KUKA KRL program: MyProgram_324().src

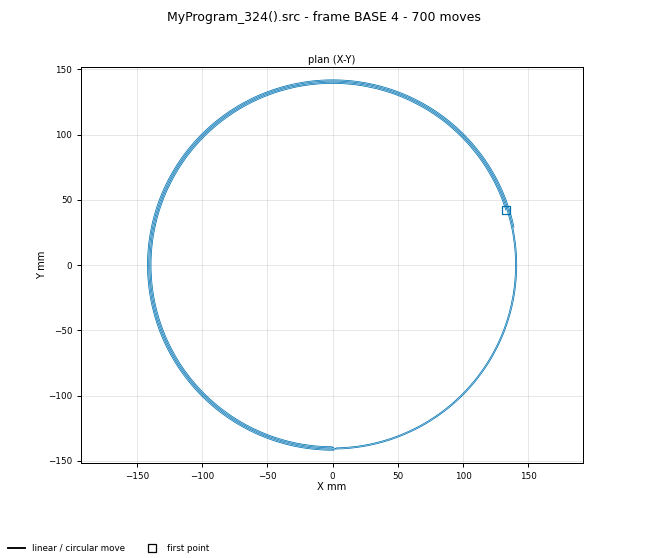
[picture p0: tool path of MyProgram_324().src in frame BASE 4, 700 of 700 moves have a stored position in this frame; points joined in program order, loops and branches not executed]
&ACCESS RVP
&REL 1
&PARAM TEMPLATE = C:\KRC\Roboter\Template\vorgabe
&PARAM EDITMASK = *
DEF MyProgram_324()
; ---- Setting reference (Base) ----
$BASE = BASE_DATA[4]

; --------------------------
; ---- Setting tool (TCP) ----
$TOOL = TOOL_DATA[3]
; --------------------------

$VEL.CP = VEL_APROX_PRINT
Startdeposition()
$VEL.CP = VEL_PRINT
LIN {X 132.7223,Y 42.0418,Z 186,A 20.4028,B 2.9301,C 0.1265,E1 3.0853,E2 432.9695} C_DIS
LIN {X 131.632,Y 45.3396,Z 186,A 21.7907,B 2.9303,C 0.1231,E1 3.0841,E2 431.5863} C_DIS
LIN {X 130.5462,Y 48.3787,Z 186,A 22.9188,B 2.9304,C 0.1215,E1 3.083,E2 430.4833} C_DIS
LIN {X 129.2167,Y 51.8236,Z 186,A 24.4942,B 2.9306,C 0.1169,E1 3.0814,E2 428.9} C_DIS
LIN {X 127.8365,Y 55.14,Z 186,A 25.9088,B 2.9307,C 0.1137,E1 3.0799,E2 427.493} C_DIS
LIN {X 126.4976,Y 58.1464,Z 186,A 27.093,B 2.9307,C 0.1118,E1 3.0786,E2 426.3301} C_DIS
LIN {X 124.9581,Y 61.3847,Z 186,A 28.6212,B 2.9309,C 0.1075,E1 3.0767,E2 424.7946} C_DIS
LIN {X 123.3471,Y 64.5607,Z 186,A 30.0105,B 2.9311,C 0.1045,E1 3.0749,E2 423.4145} C_DIS
LIN {X 121.2394,Y 68.4412,Z 186,A 31.8526,B 2.9312,C 0.0998,E1 3.0724,E2 421.5688} C_DIS
LIN {X 118.9409,Y 72.3624,Z 186,A 33.6675,B 2.9314,C 0.0957,E1 3.0698,E2 419.7604} C_DIS
LIN {X 116.4929,Y 76.2409,Z 186,A 35.4947,B 2.9314,C 0.0917,E1 3.0671,E2 417.9403} C_DIS
LIN {X 114.0875,Y 79.7952,Z 186,A 37.1739,B 2.9316,C 0.0884,E1 3.0644,E2 416.2718} C_DIS
LIN {X 111.3825,Y 83.5299,Z 186,A 38.922,B 2.9316,C 0.0853,E1 3.0616,E2 414.5422} C_DIS
LIN {X 105.7703,Y 90.5313,Z 186,A 42.3743,B 2.9318,C 0.0793,E1 3.0556,E2 411.1198} C_DIS
LIN {X 103.2392,Y 93.4068,Z 186,A 44.0814,B 2.932,C 0.0747,E1 3.0523,E2 409.3959} C_DIS
LIN {X 100.0339,Y 96.8315,Z 186,A 45.9143,B 2.932,C 0.0715,E1 3.0488,E2 407.575} C_DIS
LIN {X 96.6176,Y 100.241,Z 186,A 48.5902,B 2.9323,C 0.0615,E1 3.0433,E2 404.8112} C_DIS
LIN {X 91.8382,Y 104.6376,Z 186,A 50.3739,B 2.9323,C 0.064,E1 3.0398,E2 403.1402} C_DIS
LIN {X 88.2628,Y 107.67,Z 186,A 52.3174,B 2.9323,C 0.0602,E1 3.0356,E2 401.1947} C_DIS
LIN {X 84.6173,Y 110.5578,Z 186,A 54.1516,B 2.9323,C 0.0575,E1 3.0316,E2 399.3704} C_DIS
LIN {X 81.0366,Y 113.2086,Z 186,A 56.3803,B 2.9325,C 0.051,E1 3.0264,E2 397.0919} C_DIS
LIN {X 77.1098,Y 115.9192,Z 186,A 57.8819,B 2.9325,C 0.0516,E1 3.0231,E2 395.6486} C_DIS
LIN {X 73.3546,Y 118.3312,Z 186,A 59.6397,B 2.9325,C 0.0493,E1 3.019,E2 393.9008} C_DIS
LIN {X 69.3745,Y 120.7083,Z 186,A 61.5113,B 2.9325,C 0.0467,E1 3.0144,E2 392.0338} C_DIS
LIN {X 65.4235,Y 122.894,Z 186,A 63.1963,B 2.9325,C 0.0454,E1 3.0104,E2 390.3705} C_DIS
LIN {X 58.7576,Y 126.215,Z 186,A 66.3079,B 2.9326,C 0.0409,E1 3.0025,E2 387.2535} C_DIS
LIN {X 55.1898,Y 127.8149,Z 186,A 67.7185,B 2.9326,C 0.0405,E1 2.999,E2 385.8679} C_DIS
LIN {X 52.6155,Y 128.8975,Z 186,A 68.9895,B 2.9326,C 0.0382,E1 2.9957,E2 384.582} C_DIS
LIN {X 48.7864,Y 130.3935,Z 186,A 70.5342,B 2.9326,C 0.0374,E1 2.9917,E2 383.0558} C_DIS
LIN {X 45.2277,Y 131.6708,Z 186,A 72.3436,B 2.9327,C 0.0339,E1 2.9868,E2 381.2153} C_DIS
LIN {X 39.9443,Y 133.3707,Z 186,A 74.4722,B 2.9327,C 0.0329,E1 2.9812,E2 379.1066} C_DIS
LIN {X 36.2167,Y 134.4288,Z 186,A 75.8987,B 2.9327,C 0.0327,E1 2.9774,E2 377.7013} C_DIS
LIN {X 33.5088,Y 135.1309,Z 186,A 77.1314,B 2.9327,C 0.0312,E1 2.974,E2 376.4588} C_DIS
LIN {X 23.6749,Y 137.196,Z 186,A 81.8683,B 2.9328,C 0.0242,E1 2.9608,E2 371.6483} C_DIS
LIN {X 18.0755,Y 138.0433,Z 186,A 83.4414,B 2.9328,C 0.0283,E1 2.9567,E2 370.1703} C_DIS
LIN {X 14.3588,Y 138.4803,Z 186,A 85.0688,B 2.9328,C 0.027,E1 2.9522,E2 368.5327} C_DIS
LIN {X 10.3002,Y 138.8403,Z 186,A 86.6393,B 2.9328,C 0.027,E1 2.9478,E2 366.9759} C_DIS
LIN {X 7.1409,Y 139.0386,Z 186,A 87.9885,B 2.9328,C 0.0264,E1 2.9441,E2 365.6215} C_DIS
LIN {X 2.8453,Y 139.1938,Z 186,A 89.7701,B 2.9328,C 0.026,E1 2.9391,E2 363.8391} C_DIS
LIN {X -1.0873,Y 139.218,Z 186,A 91.4391,B 2.9328,C 0.0254,E1 2.9344,E2 362.1645} C_DIS
LIN {X -5.319,Y 139.1202,Z 186,A 92.8511,B 2.9328,C 0.0275,E1 2.9306,E2 360.794} C_DIS
LIN {X -10.208,Y 138.847,Z 186,A 95.1484,B 2.9328,C 0.0258,E1 2.9241,E2 358.4628} C_DIS
LIN {X -15.2684,Y 138.3824,Z 186,A 97.3365,B 2.9328,C 0.0255,E1 2.9179,E2 356.2638} C_DIS
LIN {X -18.8919,Y 137.9362,Z 186,A 98.9242,B 2.9328,C 0.0254,E1 2.9135,E2 354.6665} C_DIS
LIN {X -23.5933,Y 137.2096,Z 186,A 100.7482,B 2.9328,C 0.0268,E1 2.9085,E2 352.86} C_DIS
LIN {X -27.474,Y 136.4841,Z 186,A 102.3067,B 2.9328,C 0.0278,E1 2.9043,E2 351.3105} C_DIS
LIN {X -31.0328,Y 135.7188,Z 186,A 103.8636,B 2.9328,C 0.0282,E1 2.9,E2 349.7472} C_DIS
LIN {X -35.4652,Y 134.6291,Z 186,A 105.5281,B 2.9328,C 0.0305,E1 2.8956,E2 348.1102} C_DIS
LIN {X -38.2725,Y 133.8599,Z 186,A 107.0377,B 2.9328,C 0.0295,E1 2.8914,E2 346.5628} C_DIS
LIN {X -41.9969,Y 132.7366,Z 186,A 108.5373,B 2.9328,C 0.0312,E1 2.8874,E2 345.0766} C_DIS
LIN {X -45.3213,Y 131.6383,Z 186,A 110.2186,B 2.9328,C 0.0311,E1 2.8829,E2 343.3664} C_DIS
LIN {X -51.3729,Y 129.3983,Z 186,A 112.6899,B 2.9328,C 0.0344,E1 2.8765,E2 340.9196} C_DIS
LIN {X -54.8048,Y 127.9814,Z 186,A 114.2297,B 2.9327,C 0.0358,E1 2.8725,E2 339.3793} C_DIS
LIN {X -58.1767,Y 126.4836,Z 186,A 115.5667,B 2.9327,C 0.0384,E1 2.8692,E2 338.0656} C_DIS
LIN {X -60.9945,Y 125.1506,Z 186,A 117.3152,B 2.9327,C 0.0374,E1 2.8646,E2 336.2605} C_DIS
LIN {X -65.6557,Y 122.7702,Z 186,A 119.4155,B 2.9327,C 0.0403,E1 2.8595,E2 334.1683} C_DIS
LIN {X -69.1522,Y 120.8351,Z 186,A 121.2235,B 2.9327,C 0.0416,E1 2.855,E2 332.341} C_DIS
LIN {X -73.677,Y 118.1306,Z 186,A 123.2288,B 2.9326,C 0.0454,E1 2.8503,E2 330.3576} C_DIS
LIN {X -76.4881,Y 116.3301,Z 186,A 124.7057,B 2.9326,C 0.0469,E1 2.8468,E2 328.8689} C_DIS
LIN {X -80.3812,Y 113.675,Z 186,A 126.4295,B 2.9325,C 0.0508,E1 2.8429,E2 327.1733} C_DIS
LIN {X -85.7887,Y 109.6517,Z 186,A 129.4126,B 2.9325,C 0.0543,E1 2.8362,E2 324.1664} C_DIS
LIN {X -88.8265,Y 107.2052,Z 186,A 131.1719,B 2.9324,C 0.0564,E1 2.8323,E2 322.389} C_DIS
LIN {X -92.1361,Y 104.3746,Z 186,A 133.5756,B 2.9324,C 0.0569,E1 2.8271,E2 319.91} C_DIS
LIN {X -95.8456,Y 100.9798,Z 186,A 135.2159,B 2.9322,C 0.0626,E1 2.8239,E2 318.3252} C_DIS
LIN {X -98.943,Y 97.9462,Z 186,A 137.0176,B 2.9322,C 0.0659,E1 2.8203,E2 316.5226} C_DIS
LIN {X -102.1078,Y 94.6425,Z 186,A 138.7144,B 2.9321,C 0.0705,E1 2.8171,E2 314.8504} C_DIS
LIN {X -104.981,Y 91.4446,Z 186,A 140.7887,B 2.9321,C 0.0728,E1 2.8132,E2 312.7394} C_DIS
LIN {X -107.7815,Y 88.1264,Z 186,A 142.7152,B 2.9319,C 0.0761,E1 2.8097,E2 310.7967} C_DIS
LIN {X -110.7711,Y 84.3385,Z 186,A 144.7394,B 2.9319,C 0.0802,E1 2.8063,E2 308.7692} C_DIS
LIN {X -113.28,Y 80.9368,Z 186,A 146.8573,B 2.9318,C 0.0826,E1 2.8027,E2 306.6049} C_DIS
LIN {X -115.4664,Y 77.7861,Z 186,A 148.7724,B 2.9317,C 0.0849,E1 2.7997,E2 304.6482} C_DIS
LIN {X -118.3138,Y 73.3827,Z 186,A 150.3494,B 2.9315,C 0.0923,E1 2.7975,E2 303.1466} C_DIS
LIN {X -121.2066,Y 68.4995,Z 186,A 152.8996,B 2.9313,C 0.0971,E1 2.7938,E2 300.5712} C_DIS
LIN {X -123.0824,Y 65.0647,Z 186,A 154.5114,B 2.9312,C 0.101,E1 2.7917,E2 298.9603} C_DIS
LIN {X -124.7194,Y 61.8686,Z 186,A 156.0226,B 2.9311,C 0.1046,E1 2.7898,E2 297.4461} C_DIS
LIN {X -126.1022,Y 59.0017,Z 186,A 157.4751,B 2.931,C 0.1074,E1 2.7881,E2 295.9765} C_DIS
LIN {X -127.5991,Y 55.689,Z 186,A 158.8055,B 2.9308,C 0.1118,E1 2.7866,E2 294.6682} C_DIS
LIN {X -128.9832,Y 52.4027,Z 186,A 160.4995,B 2.9307,C 0.1148,E1 2.7847,E2 292.9466} C_DIS
LIN {X -130.2457,Y 49.1811,Z 186,A 162.0157,B 2.9305,C 0.1182,E1 2.7832,E2 291.4197} C_DIS
LIN {X -131.4915,Y 45.7449,Z 186,A 163.5273,B 2.9304,C 0.1221,E1 2.7818,E2 289.9083} C_DIS
LIN {X -132.4989,Y 42.741,Z 186,A 164.9566,B 2.9302,C 0.1252,E1 2.7805,E2 288.464} C_DIS
LIN {X -133.544,Y 39.3531,Z 186,A 166.487,B 2.9301,C 0.1288,E1 2.7793,E2 286.9256} C_DIS
LIN {X -134.4876,Y 35.9962,Z 186,A 167.975,B 2.9299,C 0.1325,E1 2.7782,E2 285.4318} C_DIS
LIN {X -135.4954,Y 32.0004,Z 186,A 169.8584,B 2.9297,C 0.1365,E1 2.7769,E2 283.5256} C_DIS
LIN {X -136.2453,Y 28.643,Z 186,A 171.4142,B 2.9296,C 0.1399,E1 2.776,E2 281.953} C_DIS
LIN {X -137.073,Y 24.3655,Z 186,A 173.1645,B 2.9293,C 0.145,E1 2.7751,E2 280.2093} C_DIS
LIN {X -137.8774,Y 19.304,Z 186,A 175.9731,B 2.9292,C 0.1485,E1 2.774,E2 277.3117} C_DIS
LIN {X -138.4947,Y 14.2251,Z 186,A 177.6797,B 2.9288,C 0.1558,E1 2.7735,E2 275.6584} C_DIS
LIN {X -138.8515,Y 10.1468,Z 186,A 179.1361,B 2.9285,C 0.1613,E1 2.7731,E2 274.2326} C_DIS
LIN {X -139.1571,Y 4.2614,Z 186,A -178.1292,B 2.9282,C 0.1671,E1 2.7728,E2 271.4597} C_DIS
LIN {X -139.1979,Y -2.5987,Z 186,A -175.1607,B 2.9277,C 0.1745,E1 2.7728,E2 268.4743} C_DIS
LIN {X -138.9299,Y -9.0223,Z 186,A -172.252,B 2.9273,C 0.181,E1 2.7732,E2 265.5331} C_DIS
LIN {X -138.4477,Y -14.6613,Z 186,A -169.9308,B 2.9269,C 0.1876,E1 2.7738,E2 263.2143} C_DIS
LIN {X -138.0238,Y -18.2243,Z 186,A -168.3737,B 2.9267,C 0.1914,E1 2.7743,E2 261.6475} C_DIS
LIN {X -137.1804,Y -23.7653,Z 186,A -165.8389,B 2.9263,C 0.197,E1 2.7755,E2 259.0843} C_DIS
LIN {X -136.3999,Y -27.8879,Z 186,A -164.1464,B 2.926,C 0.2018,E1 2.7764,E2 257.3971} C_DIS
LIN {X -135.6392,Y -31.3814,Z 186,A -162.4754,B 2.9257,C 0.2051,E1 2.7774,E2 255.7008} C_DIS
LIN {X -134.6193,Y -35.5023,Z 186,A -160.7508,B 2.9254,C 0.21,E1 2.7786,E2 253.98} C_DIS
LIN {X -133.6857,Y -38.8692,Z 186,A -159.2487,B 2.9251,C 0.2136,E1 2.7798,E2 252.4702} C_DIS
LIN {X -132.7391,Y -41.989,Z 186,A -157.9755,B 2.9249,C 0.2174,E1 2.7808,E2 251.2067} C_DIS
LIN {X -131.652,Y -45.2818,Z 186,A -156.5515,B 2.9246,C 0.2212,E1 2.7821,E2 249.7838} C_DIS
LIN {X -129.709,Y -50.5783,Z 186,A -153.8693,B 2.9242,C 0.2259,E1 2.7847,E2 247.0551} C_DIS
LIN {X -128.6254,Y -53.2752,Z 186,A -152.4667,B 2.924,C 0.2282,E1 2.7863,E2 245.6256} C_DIS
LIN {X -126.553,Y -58.0266,Z 186,A -150.3996,B 2.9236,C 0.2338,E1 2.7886,E2 243.5682} C_DIS
LIN {X -125.0099,Y -61.2796,Z 186,A -148.8804,B 2.9233,C 0.2374,E1 2.7904,E2 242.0446} C_DIS
LIN {X -123.6519,Y -63.9802,Z 186,A -147.5183,B 2.9231,C 0.24,E1 2.7922,E2 240.6673} C_DIS
LIN {X -119.8995,Y -70.7624,Z 186,A -144.2009,B 2.9225,C 0.2471,E1 2.7968,E2 237.3341} C_DIS
LIN {X -117.3139,Y -74.9705,Z 186,A -142.0411,B 2.9221,C 0.2513,E1 2.8,E2 235.158} C_DIS
LIN {X -114.7566,Y -78.8292,Z 186,A -140.0835,B 2.9218,C 0.2554,E1 2.8031,E2 233.1939} C_DIS
LIN {X -112.8116,Y -81.5885,Z 186,A -138.2374,B 2.9217,C 0.2565,E1 2.8062,E2 231.2867} C_DIS
LIN {X -110.2703,Y -84.9925,Z 186,A -136.7891,B 2.9212,C 0.2616,E1 2.8086,E2 229.8793} C_DIS
LIN {X -107.4976,Y -88.4735,Z 186,A -134.8803,B 2.9209,C 0.2651,E1 2.8119,E2 227.9605} C_DIS
LIN {X -104.5729,Y -91.9119,Z 186,A -133.2398,B 2.9205,C 0.2699,E1 2.8149,E2 226.3495} C_DIS
LIN {X -102.4762,Y -94.243,Z 186,A -131.6371,B 2.9204,C 0.271,E1 2.818,E2 224.705} C_DIS
LIN {X -99.0053,Y -97.8835,Z 186,A -129.2575,B 2.9201,C 0.2735,E1 2.8227,E2 222.284} C_DIS
LIN {X -96.5135,Y -100.3416,Z 186,A -127.9872,B 2.9198,C 0.277,E1 2.8252,E2 221.0369} C_DIS
LIN {X -93.1987,Y -103.4277,Z 186,A -126.0443,B 2.9195,C 0.28,E1 2.8292,E2 219.0834} C_DIS
LIN {X -89.6587,Y -106.5105,Z 186,A -124.0623,B 2.9192,C 0.283,E1 2.8335,E2 217.0948} C_DIS
LIN {X -86,Y -109.4857,Z 186,A -122.1302,B 2.9189,C 0.2863,E1 2.8377,E2 215.164} C_DIS
LIN {X -77.5113,Y -115.6511,Z 186,A -117.9132,B 2.9182,C 0.2934,E1 2.8472,E2 210.961} C_DIS
LIN {X -74.5846,Y -117.5601,Z 186,A -116.1603,B 2.9182,C 0.2937,E1 2.8514,E2 209.1654} C_DIS
LIN {X -70.7202,Y -119.9243,Z 186,A -114.2581,B 2.918,C 0.2959,E1 2.856,E2 207.2579} C_DIS
LIN {X -66.4872,Y -122.3218,Z 186,A -111.2975,B 2.9183,C 0.2929,E1 2.8636,E2 204.1656} C_DIS
LIN {X -60.0963,Y -125.5826,Z 186,A -109.3331,B 2.9174,C 0.3018,E1 2.8682,E2 202.3365} C_DIS
LIN {X -56.0089,Y -127.4608,Z 186,A -107.4407,B 2.9172,C 0.3034,E1 2.873,E2 200.4383} C_DIS
LIN {X -52.4435,Y -128.9668,Z 186,A -105.8095,B 2.9171,C 0.3047,E1 2.8773,E2 198.8016} C_DIS
LIN {X -48.4538,Y -130.5181,Z 186,A -103.8163,B 2.9171,C 0.3047,E1 2.8826,E2 196.7763} C_DIS
LIN {X -44.2579,Y -131.9997,Z 186,A -102.3244,B 2.9167,C 0.3082,E1 2.8864,E2 195.3304} C_DIS
LIN {X -41.04,Y -133.0354,Z 186,A -100.7788,B 2.9167,C 0.3082,E1 2.8906,E2 193.7634} C_DIS
LIN {X -37.7743,Y -133.9992,Z 186,A -99.5511,B 2.9165,C 0.3102,E1 2.8938,E2 192.559} C_DIS
LIN {X -34.537,Y -134.8699,Z 186,A -97.2089,B 2.917,C 0.3048,E1 2.9005,E2 190.0842} C_DIS
LIN {X -28.8904,Y -136.1919,Z 186,A -95.4264,B 2.9165,C 0.3097,E1 2.9051,E2 188.3843} C_DIS
LIN {X -23.7358,Y -137.1857,Z 186,A -93.3501,B 2.9164,C 0.311,E1 2.9108,E2 186.3188} C_DIS
LIN {X -19.9134,Y -137.7903,Z 186,A -91.8953,B 2.9163,C 0.3123,E1 2.9148,E2 184.8822} C_DIS
LIN {X -16.6105,Y -138.2273,Z 186,A -90.3853,B 2.9163,C 0.3116,E1 2.919,E2 183.3527} C_DIS
LIN {X -13.0475,Y -138.6092,Z 186,A -88.8614,B 2.9163,C 0.3115,E1 2.9233,E2 181.8214} C_DIS
LIN {X -8.7396,Y -138.9473,Z 186,A -87.083,B 2.9163,C 0.3115,E1 2.9283,E2 180.0424} C_DIS
LIN {X -4.337,Y -139.155,Z 186,A -85.2848,B 2.9163,C 0.3115,E1 2.9333,E2 178.2455} C_DIS
LIN {X -0.6821,Y -139.2202,Z 186,A -83.7898,B 2.9163,C 0.3113,E1 2.9375,E2 176.7511} C_DIS
LIN {X -0.6821,Y -139.2202,Z 186,A -83.7898,B 2.9163,C 0.3113,E1 2.9375,E2 176.7511} C_DIS
Enddeposition()
LIN {X 1.0073,Y -140.1176,Z 186,A -83.0914,B 2.892,C 0.3118,E1 2.9151,E2 176.0888} C_DIS
Startdeposition()
$VEL.CP = VEL_PRINT
LIN {X -2.8203,Y -140.0942,Z 186,A -85.3593,B 2.8914,C 0.317,E1 2.9085,E2 178.4541} C_DIS
LIN {X -7.0046,Y -139.9465,Z 186,A -86.9368,B 2.8915,C 0.3162,E1 2.9041,E2 180.014} C_DIS
LIN {X -10.1238,Y -139.7554,Z 186,A -88.277,B 2.8915,C 0.3166,E1 2.9004,E2 181.3632} C_DIS
LIN {X -14.2012,Y -139.4023,Z 186,A -90.0662,B 2.8915,C 0.3172,E1 2.8953,E2 183.169} C_DIS
LIN {X -18.1624,Y -138.9394,Z 186,A -91.5726,B 2.8915,C 0.3161,E1 2.8912,E2 184.659} C_DIS
LIN {X -21.6584,Y -138.4377,Z 186,A -93.0477,B 2.8915,C 0.316,E1 2.8871,E2 186.1389} C_DIS
LIN {X -26.4802,Y -137.5967,Z 186,A -95.0602,B 2.8916,C 0.3154,E1 2.8816,E2 188.1536} C_DIS
LIN {X -30.6439,Y -136.7307,Z 186,A -97.0086,B 2.8916,C 0.316,E1 2.8762,E2 190.1311} C_DIS
LIN {X -38.0299,Y -134.8621,Z 186,A -99.9566,B 2.8919,C 0.3133,E1 2.8683,E2 193.0572} C_DIS
LIN {X -42.2307,Y -133.6066,Z 186,A -101.7675,B 2.8919,C 0.3122,E1 2.8634,E2 194.8711} C_DIS
LIN {X -49.1907,Y -131.203,Z 186,A -104.7675,B 2.8922,C 0.3098,E1 2.8555,E2 197.8703} C_DIS
LIN {X -52.5755,Y -129.8838,Z 186,A -106.3058,B 2.8923,C 0.3088,E1 2.8515,E2 199.4161} C_DIS
LIN {X -55.9211,Y -128.4791,Z 186,A -107.8545,B 2.8924,C 0.3078,E1 2.8475,E2 200.9739} C_DIS
LIN {X -59.073,Y -127.0606,Z 186,A -109.2324,B 2.8926,C 0.3062,E1 2.844,E2 202.3472} C_DIS
LIN {X -61.9775,Y -125.6691,Z 186,A -110.9944,B 2.8926,C 0.3072,E1 2.8394,E2 204.1697} C_DIS
LIN {X -65.5403,Y -123.8491,Z 186,A -112.3239,B 2.8929,C 0.3036,E1 2.8362,E2 205.458} C_DIS
LIN {X -69.6738,Y -121.5736,Z 186,A -114.3235,B 2.8931,C 0.3016,E1 2.8313,E2 207.4673} C_DIS
LIN {X -73.6489,Y -119.2079,Z 186,A -116.2465,B 2.8933,C 0.2993,E1 2.8267,E2 209.3948} C_DIS
LIN {X -77.3828,Y -116.8184,Z 186,A -118.1408,B 2.8936,C 0.2972,E1 2.8222,E2 211.3001} C_DIS
LIN {X -82.8133,Y -113.0326,Z 186,A -121.0194,B 2.8939,C 0.294,E1 2.8156,E2 214.2019} C_DIS
LIN {X -86.9995,Y -109.8439,Z 186,A -123.1378,B 2.8942,C 0.2904,E1 2.811,E2 216.3157} C_DIS
LIN {X -90.5099,Y -106.9698,Z 186,A -125.2597,B 2.8944,C 0.2885,E1 2.8063,E2 218.4735} C_DIS
LIN {X -93.182,Y -104.6507,Z 186,A -126.5493,B 2.8948,C 0.2853,E1 2.8037,E2 219.7417} C_DIS
LIN {X -99.3475,Y -98.8158,Z 186,A -130.0753,B 2.8953,C 0.2791,E1 2.7966,E2 223.2747} C_DIS
LIN {X -102.3742,Y -95.6769,Z 186,A -131.9754,B 2.8956,C 0.2762,E1 2.7929,E2 225.1904} C_DIS
LIN {X -106.548,Y -91.0061,Z 186,A -134.4714,B 2.8961,C 0.2707,E1 2.7883,E2 227.6771} C_DIS
LIN {X -108.9363,Y -88.133,Z 186,A -137.1963,B 2.896,C 0.2727,E1 2.7833,E2 230.5608} C_DIS
LIN {X -113.5466,Y -82.1078,Z 186,A -139.3898,B 2.8969,C 0.262,E1 2.7798,E2 232.6331} C_DIS
LIN {X -116.1588,Y -78.3689,Z 186,A -141.3574,B 2.8973,C 0.2583,E1 2.7767,E2 234.6139} C_DIS
LIN {X -118.6593,Y -74.5284,Z 186,A -143.1364,B 2.8977,C 0.2536,E1 2.774,E2 236.3797} C_DIS
LIN {X -120.5144,Y -71.4903,Z 186,A -145.0644,B 2.8978,C 0.252,E1 2.7711,E2 238.3701} C_DIS
LIN {X -122.2481,Y -68.4828,Z 186,A -146.4171,B 2.8981,C 0.2484,E1 2.7693,E2 239.7134} C_DIS
LIN {X -124.3266,Y -64.6308,Z 186,A -148.2148,B 2.8985,C 0.244,E1 2.767,E2 241.5115} C_DIS
LIN {X -126.3123,Y -60.6565,Z 186,A -150.0063,B 2.8989,C 0.2394,E1 2.7647,E2 243.299} C_DIS
LIN {X -127.8057,Y -57.4429,Z 186,A -151.6407,B 2.8991,C 0.2365,E1 2.7628,E2 244.9572} C_DIS
LIN {X -129.3909,Y -53.7772,Z 186,A -153.1363,B 2.8995,C 0.2318,E1 2.7612,E2 246.4339} C_DIS
LIN {X -130.9844,Y -49.7724,Z 186,A -155.3764,B 2.8997,C 0.229,E1 2.7589,E2 248.7362} C_DIS
LIN {X -132.1779,Y -46.5121,Z 186,A -156.4594,B 2.9001,C 0.224,E1 2.7579,E2 249.7743} C_DIS
LIN {X -133.0781,Y -43.8676,Z 186,A -157.7354,B 2.9003,C 0.2215,E1 2.7568,E2 251.0675} C_DIS
LIN {X -134.2034,Y -40.2984,Z 186,A -159.4915,B 2.9006,C 0.2183,E1 2.7553,E2 252.8525} C_DIS
LIN {X -135.3756,Y -36.1585,Z 186,A -161.2152,B 2.9009,C 0.2134,E1 2.754,E2 254.5705} C_DIS
LIN {X -136.2522,Y -32.7009,Z 186,A -162.7135,B 2.9012,C 0.2096,E1 2.753,E2 256.0733} C_DIS
LIN {X -137.0113,Y -29.3591,Z 186,A -164.2143,B 2.9015,C 0.2061,E1 2.7521,E2 257.5864} C_DIS
LIN {X -137.8186,Y -25.307,Z 186,A -166.7114,B 2.9015,C 0.2043,E1 2.7508,E2 260.1875} C_DIS
LIN {X -138.7087,Y -19.8477,Z 186,A -168.0276,B 2.9022,C 0.1947,E1 2.7503,E2 261.3795} C_DIS
LIN {X -139.1085,Y -16.8203,Z 186,A -170.2463,B 2.9022,C 0.1946,E1 2.7495,E2 263.7236} C_DIS
LIN {X -139.6024,Y -12.0542,Z 186,A -171.4913,B 2.9028,C 0.1867,E1 2.7492,E2 264.8749} C_DIS
LIN {X -140.0378,Y -4.8813,Z 186,A -174.7473,B 2.9032,C 0.1795,E1 2.7487,E2 268.1706} C_DIS
LIN {X -140.114,Y -1.6302,Z 186,A -176.6869,B 2.9033,C 0.1778,E1 2.7486,E2 270.188} C_DIS
LIN {X -140.1002,Y 2.4604,Z 186,A -177.8971,B 2.9037,C 0.1716,E1 2.7486,E2 271.3376} C_DIS
LIN {X -139.7549,Y 10.1308,Z 186,A 178.8114,B 2.9042,C 0.1633,E1 2.7491,E2 274.6468} C_DIS
LIN {X -138.9275,Y 18.2534,Z 186,A 174.7575,B 2.9046,C 0.1563,E1 2.7504,E2 278.7901} C_DIS
LIN {X -138.3187,Y 22.4138,Z 186,A 173.4853,B 2.9049,C 0.15,E1 2.7509,E2 280.0041} C_DIS
LIN {X -137.5893,Y 26.5188,Z 186,A 171.6337,B 2.9051,C 0.1458,E1 2.7518,E2 281.8732} C_DIS
LIN {X -136.4611,Y 31.824,Z 186,A 169.3535,B 2.9054,C 0.1399,E1 2.7532,E2 284.1598} C_DIS
LIN {X -135.8128,Y 34.4801,Z 186,A 168.0816,B 2.9055,C 0.1374,E1 2.754,E2 285.4506} C_DIS
LIN {X -134.8776,Y 37.9746,Z 186,A 166.561,B 2.9057,C 0.1335,E1 2.7552,E2 286.9753} C_DIS
LIN {X -133.8797,Y 41.356,Z 186,A 165.0431,B 2.9059,C 0.1299,E1 2.7564,E2 288.5019} C_DIS
LIN {X -132.8695,Y 44.4938,Z 186,A 163.5863,B 2.906,C 0.1267,E1 2.7577,E2 289.9716} C_DIS
LIN {X -131.6328,Y 48.0318,Z 186,A 162.0329,B 2.9062,C 0.1227,E1 2.7591,E2 291.5265} C_DIS
LIN {X -130.5108,Y 50.9993,Z 186,A 160.6348,B 2.9062,C 0.1197,E1 2.7605,E2 292.9363} C_DIS
LIN {X -129.1805,Y 54.281,Z 186,A 159.1523,B 2.9064,C 0.1161,E1 2.7621,E2 294.4222} C_DIS
LIN {X -127.7897,Y 57.4787,Z 186,A 157.6404,B 2.9066,C 0.1127,E1 2.7638,E2 295.9439} C_DIS
LIN {X -126.244,Y 60.7995,Z 186,A 156.093,B 2.9067,C 0.1091,E1 2.7657,E2 297.4964} C_DIS
LIN {X -124.7604,Y 63.7873,Z 186,A 154.6494,B 2.9068,C 0.106,E1 2.7675,E2 298.949} C_DIS
LIN {X -123.0275,Y 67.0726,Z 186,A 152.9761,B 2.9069,C 0.1028,E1 2.7698,E2 300.6406} C_DIS
LIN {X -120.9497,Y 70.7512,Z 186,A 151.3206,B 2.9071,C 0.0984,E1 2.772,E2 302.2858} C_DIS
LIN {X -119.0618,Y 73.8837,Z 186,A 149.0959,B 2.9071,C 0.0976,E1 2.7755,E2 304.6004} C_DIS
LIN {X -116.3995,Y 78.0105,Z 186,A 147.5398,B 2.9073,C 0.0912,E1 2.7778,E2 306.0987} C_DIS
LIN {X -114.4773,Y 80.8049,Z 186,A 146.1663,B 2.9074,C 0.088,E1 2.7799,E2 307.4694} C_DIS
LIN {X -112.085,Y 84.0928,Z 186,A 144.4493,B 2.9075,C 0.0846,E1 2.7828,E2 309.1921} C_DIS
LIN {X -109.706,Y 87.1728,Z 186,A 142.4375,B 2.9075,C 0.0828,E1 2.7864,E2 311.2549} C_DIS
LIN {X -107.4678,Y 89.9177,Z 186,A 140.3627,B 2.9075,C 0.0822,E1 2.7903,E2 313.4059} C_DIS
LIN {X -103.1556,Y 94.8336,Z 186,A 138.8315,B 2.9079,C 0.0721,E1 2.7929,E2 314.7937} C_DIS
LIN {X -99.7013,Y 98.4597,Z 186,A 136.251,B 2.9079,C 0.0703,E1 2.798,E2 317.4391} C_DIS
LIN {X -96.4124,Y 101.6822,Z 186,A 134.12,B 2.9079,C 0.0678,E1 2.8023,E2 319.5994} C_DIS
LIN {X -93.9584,Y 103.9533,Z 186,A 133.0252,B 2.9081,C 0.0641,E1 2.8045,E2 320.6595} C_DIS
LIN {X -90.9705,Y 106.5783,Z 186,A 131.2328,B 2.9081,C 0.062,E1 2.8083,E2 322.4712} C_DIS
LIN {X -87.5,Y 109.4455,Z 186,A 129.3243,B 2.9081,C 0.0592,E1 2.8125,E2 324.3868} C_DIS
LIN {X -83.0265,Y 112.8765,Z 186,A 127.0447,B 2.9082,C 0.0553,E1 2.8176,E2 326.6615} C_DIS
LIN {X -80.4773,Y 114.7084,Z 186,A 125.6391,B 2.9082,C 0.0539,E1 2.8208,E2 328.0814} C_DIS
LIN {X -76.0708,Y 117.6767,Z 186,A 123.523,B 2.9083,C 0.0505,E1 2.8257,E2 330.189} C_DIS
LIN {X -69.6537,Y 121.585,Z 186,A 120.5702,B 2.9084,C 0.0457,E1 2.8327,E2 333.1251} C_DIS
LIN {X -66.865,Y 123.1407,Z 186,A 118.9491,B 2.9084,C 0.0457,E1 2.8368,E2 334.7842} C_DIS
LIN {X -63.6921,Y 124.8089,Z 186,A 116.8207,B 2.9084,C 0.0472,E1 2.8423,E2 336.9926} C_DIS
LIN {X -58.6521,Y 127.2552,Z 186,A 115.2003,B 2.9084,C 0.0413,E1 2.8462,E2 338.5297} C_DIS
LIN {X -55.5464,Y 128.6411,Z 186,A 113.3543,B 2.9084,C 0.0422,E1 2.8511,E2 340.4305} C_DIS
LIN {X -51.6471,Y 130.258,Z 186,A 112.0559,B 2.9085,C 0.0384,E1 2.8543,E2 341.6756} C_DIS
LIN {X -45.7089,Y 132.4564,Z 186,A 109.4422,B 2.9085,C 0.0363,E1 2.8612,E2 344.2907} C_DIS
LIN {X -42.6797,Y 133.4631,Z 186,A 108.0307,B 2.9085,C 0.0359,E1 2.8649,E2 345.7145} C_DIS
LIN {X -38.6935,Y 134.6748,Z 186,A 105.9805,B 2.9085,C 0.0367,E1 2.8706,E2 347.8062} C_DIS
LIN {X -35.0744,Y 135.6619,Z 186,A 104.8968,B 2.9085,C 0.0333,E1 2.8733,E2 348.8339} C_DIS
LIN {X -31.1063,Y 136.625,Z 186,A 103.121,B 2.9085,C 0.033,E1 2.8782,E2 350.6218} C_DIS
LIN {X -27.6399,Y 137.3686,Z 186,A 101.6275,B 2.9085,C 0.0326,E1 2.8823,E2 352.1198} C_DIS
LIN {X -19.4073,Y 138.7716,Z 186,A 98.2081,B 2.9085,C 0.0315,E1 2.8918,E2 355.5382} C_DIS
LIN {X -15.2807,Y 139.2861,Z 186,A 96.3935,B 2.9085,C 0.0319,E1 2.8968,E2 357.3659} C_DIS
LIN {X -9.1316,Y 139.8247,Z 186,A 94.0918,B 2.9086,C 0.0303,E1 2.9032,E2 359.6392} C_DIS
LIN {X -5.475,Y 140.0147,Z 186,A 92.504,B 2.9086,C 0.0308,E1 2.9076,E2 361.2375} C_DIS
LIN {X -1.7806,Y 140.1115,Z 186,A 90.8716,B 2.9086,C 0.0317,E1 2.9122,E2 362.8841} C_DIS
LIN {X 2.2977,Y 140.1029,Z 186,A 89.283,B 2.9086,C 0.0315,E1 2.9166,E2 364.4623} C_DIS
LIN {X 6.5026,Y 139.9717,Z 186,A 87.5403,B 2.9086,C 0.032,E1 2.9215,E2 366.2072} C_DIS
LIN {X 10.1851,Y 139.7509,Z 186,A 86.1055,B 2.9086,C 0.032,E1 2.9255,E2 367.6322} C_DIS
LIN {X 13.5142,Y 139.4684,Z 186,A 84.7785,B 2.9086,C 0.0323,E1 2.9292,E2 368.954} C_DIS
LIN {X 16.8125,Y 139.1094,Z 186,A 83.3856,B 2.9086,C 0.0331,E1 2.933,E2 370.3509} C_DIS
LIN {X 20.7808,Y 138.5735,Z 186,A 81.6286,B 2.9086,C 0.0348,E1 2.938,E2 372.122} C_DIS
LIN {X 24.9414,Y 137.8841,Z 186,A 80.0662,B 2.9086,C 0.0348,E1 2.9422,E2 373.6639} C_DIS
LIN {X 28.7642,Y 137.1389,Z 186,A 78.398,B 2.9086,C 0.0364,E1 2.9468,E2 375.341} C_DIS
LIN {X 34.8216,Y 135.7261,Z 186,A 76.0373,B 2.9086,C 0.037,E1 2.9532,E2 377.6786} C_DIS
LIN {X 37.7562,Y 134.9387,Z 186,A 74.7605,B 2.9086,C 0.0384,E1 2.9566,E2 378.9593} C_DIS
LIN {X 41.0365,Y 133.9775,Z 186,A 72.7793,B 2.9084,C 0.0439,E1 2.9621,E2 381.0117} C_DIS
LIN {X 45.9497,Y 132.3729,Z 186,A 71.3347,B 2.9084,C 0.0412,E1 2.9657,E2 382.3738} C_DIS
LIN {X 49.3723,Y 131.135,Z 186,A 69.8501,B 2.9084,C 0.0427,E1 2.9696,E2 383.8578} C_DIS
LIN {X 52.5122,Y 129.9093,Z 186,A 68.4786,B 2.9084,C 0.0443,E1 2.9732,E2 385.2282} C_DIS
LIN {X 55.9067,Y 128.4853,Z 186,A 67.0199,B 2.9084,C 0.0458,E1 2.9769,E2 386.6809} C_DIS
LIN {X 59.6622,Y 126.7873,Z 186,A 64.9469,B 2.9084,C 0.0509,E1 2.9823,E2 388.8016} C_DIS
LIN {X 63.296,Y 125.0105,Z 186,A 63.7666,B 2.9084,C 0.0495,E1 2.9851,E2 389.9232} C_DIS
LIN {X 66.2429,Y 123.4762,Z 186,A 62.3458,B 2.9083,C 0.0519,E1 2.9886,E2 391.3517} C_DIS
LIN {X 70.384,Y 121.1636,Z 186,A 60.4785,B 2.9083,C 0.0542,E1 2.9931,E2 393.2099} C_DIS
LIN {X 74.0809,Y 118.9391,Z 186,A 58.7482,B 2.9083,C 0.0567,E1 2.9972,E2 394.9359} C_DIS
LIN {X 77.9035,Y 116.4713,Z 186,A 56.7162,B 2.9081,C 0.0612,E1 3.002,E2 396.9892} C_DIS
LIN {X 80.7684,Y 114.5031,Z 186,A 55.59,B 2.9081,C 0.0612,E1 3.0045,E2 398.0788} C_DIS
LIN {X 84.2612,Y 111.9579,Z 186,A 53.8305,B 2.9081,C 0.0642,E1 3.0085,E2 399.8374} C_DIS
LIN {X 87.7944,Y 109.2093,Z 186,A 52.0517,B 2.908,C 0.0671,E1 3.0124,E2 401.6098} C_DIS
LIN {X 90.5408,Y 106.9436,Z 186,A 50.6985,B 2.908,C 0.069,E1 3.0152,E2 402.9503} C_DIS
LIN {X 94.7809,Y 103.204,Z 186,A 48.2327,B 2.9078,C 0.0748,E1 3.0204,E2 405.4356} C_DIS
LIN {X 97.2214,Y 100.9089,Z 186,A 47.0627,B 2.9078,C 0.0758,E1 3.0227,E2 406.5808} C_DIS
LIN {X 100.4442,Y 97.7014,Z 186,A 45.2766,B 2.9077,C 0.079,E1 3.0262,E2 408.358} C_DIS
LIN {X 103.505,Y 94.4529,Z 186,A 43.4994,B 2.9076,C 0.0825,E1 3.0296,E2 410.1295} C_DIS
LIN {X 105.9389,Y 91.7146,Z 186,A 42.0828,B 2.9076,C 0.085,E1 3.0321,E2 411.5362} C_DIS
LIN {X 109.786,Y 87.0711,Z 186,A 39.7594,B 2.9074,C 0.0893,E1 3.0362,E2 413.8421} C_DIS
LIN {X 112.085,Y 84.0928,Z 186,A 38.2173,B 2.9073,C 0.0928,E1 3.0388,E2 415.3851} C_DIS
LIN {X 114.795,Y 80.3539,Z 186,A 36.3996,B 2.9072,C 0.0966,E1 3.0418,E2 417.1945} C_DIS
LIN {X 117.3488,Y 76.5759,Z 186,A 34.6076,B 2.907,C 0.1004,E1 3.0445,E2 418.9778} C_DIS
LIN {X 119.8062,Y 72.6706,Z 186,A 32.8142,B 2.9069,C 0.1041,E1 3.0471,E2 420.76} C_DIS
LIN {X 122.1328,Y 68.6883,Z 186,A 31.0315,B 2.9068,C 0.1078,E1 3.0496,E2 422.5301} C_DIS
LIN {X 124.2212,Y 64.8315,Z 186,A 29.4036,B 2.9067,C 0.1108,E1 3.0517,E2 424.1375} C_DIS
LIN {X 125.8531,Y 61.6045,Z 186,A 27.9865,B 2.9065,C 0.1139,E1 3.0535,E2 425.5473} C_DIS
LIN {X 127.2965,Y 58.5628,Z 186,A 26.646,B 2.9065,C 0.1171,E1 3.055,E2 426.8837} C_DIS
LIN {X 128.7275,Y 55.3466,Z 186,A 25.2431,B 2.9063,C 0.1205,E1 3.0566,E2 428.2826} C_DIS
LIN {X 130.4291,Y 51.2095,Z 186,A 23.4905,B 2.9061,C 0.1246,E1 3.0584,E2 430.0262} C_DIS
LIN {X 131.7711,Y 47.6481,Z 186,A 22.0604,B 2.906,C 0.1276,E1 3.0598,E2 431.4407} C_DIS
LIN {X 132.8864,Y 44.4432,Z 186,A 20.6842,B 2.9058,C 0.1312,E1 3.061,E2 432.8162} C_DIS
LIN {X 134.0315,Y 40.86,Z 186,A 19.2077,B 2.9056,C 0.1347,E1 3.0623,E2 434.2855} C_DIS
LIN {X 135.6796,Y 35.0046,Z 186,A 16.9816,B 2.9054,C 0.139,E1 3.0639,E2 436.4792} C_DIS
LIN {X 136.5324,Y 31.512,Z 186,A 15.1481,B 2.9051,C 0.1465,E1 3.0651,E2 438.3603} C_DIS
LIN {X 137.2928,Y 28.0124,Z 186,A 13.7177,B 2.9049,C 0.1502,E1 3.0659,E2 439.7871} C_DIS
LIN {X 138.0122,Y 24.2255,Z 186,A 12.4853,B 2.9049,C 0.1513,E1 3.0665,E2 440.976} C_DIS
LIN {X 138.7697,Y 19.4206,Z 186,A 10.558,B 2.9046,C 0.1563,E1 3.0673,E2 442.8965} C_DIS
LIN {X 139.3092,Y 15.0667,Z 186,A 8.9556,B 2.9044,C 0.1594,E1 3.0678,E2 444.4751} C_DIS
LIN {X 139.675,Y 11.1945,Z 186,A 7.326,B 2.9041,C 0.1643,E1 3.0682,E2 446.1108} C_DIS
LIN {X 139.943,Y 7.0726,Z 186,A 5.816,B 2.9039,C 0.1673,E1 3.0684,E2 447.5985} C_DIS
LIN {X 140.0789,Y 3.4872,Z 186,A 4.3331,B 2.9037,C 0.1716,E1 3.0685,E2 449.0844} C_DIS
LIN {X 140.1216,Y -0.6105,Z 186,A 2.7555,B 2.9035,C 0.1753,E1 3.0685,E2 450.6503} C_DIS
LIN {X 140.0521,Y -4.4514,Z 186,A 1.2327,B 2.9032,C 0.1793,E1 3.0685,E2 452.1679} C_DIS
LIN {X 139.8502,Y -8.7178,Z 186,A -0.3532,B 2.903,C 0.1826,E1 3.0682,E2 453.7339} C_DIS
LIN {X 139.5075,Y -13.107,Z 186,A -2.0932,B 2.9027,C 0.1871,E1 3.0678,E2 455.4673} C_DIS
LIN {X 139.121,Y -16.715,Z 186,A -3.4498,B 2.9026,C 0.19,E1 3.0674,E2 456.8081} C_DIS
LIN {X 138.6028,Y -20.5827,Z 186,A -4.9386,B 2.9023,C 0.1934,E1 3.0668,E2 458.284} C_DIS
LIN {X 138.1715,Y -23.2964,Z 186,A -6.0873,B 2.9021,C 0.1968,E1 3.0663,E2 459.4369} C_DIS
LIN {X 136.6474,Y -31.0085,Z 186,A -9.8818,B 2.9011,C 0.2113,E1 3.064,E2 463.3096} C_DIS
LIN {X 135.1293,Y -37.0746,Z 186,A -11.4979,B 2.9012,C 0.2092,E1 3.063,E2 464.8041} C_DIS
LIN {X 133.8971,Y -41.2993,Z 186,A -13.3419,B 2.9008,C 0.2145,E1 3.0615,E2 466.6552} C_DIS
LIN {X 132.5147,Y -45.5408,Z 186,A -15.3839,B 2.9003,C 0.2216,E1 3.0597,E2 468.7275} C_DIS
LIN {X 131.2253,Y -49.1312,Z 186,A -16.2197,B 2.9005,C 0.2187,E1 3.059,E2 469.4684} C_DIS
LIN {X 129.8729,Y -52.6026,Z 186,A -18.0178,B 2.9,C 0.2254,E1 3.0571,E2 471.3042} C_DIS
LIN {X 128.2347,Y -56.4838,Z 186,A -20.0646,B 2.8994,C 0.233,E1 3.0547,E2 473.3955} C_DIS
LIN {X 126.4821,Y -60.301,Z 186,A -20.9998,B 2.8997,C 0.23,E1 3.0538,E2 474.2278} C_DIS
LIN {X 124.6085,Y -64.0856,Z 186,A -23.4741,B 2.8987,C 0.2415,E1 3.0505,E2 476.8032} C_DIS
LIN {X 122.218,Y -68.5367,Z 186,A -24.9859,B 2.8987,C 0.2415,E1 3.0485,E2 478.243} C_DIS
LIN {X 119.8831,Y -72.5433,Z 186,A -26.7888,B 2.8984,C 0.2452,E1 3.046,E2 480.0349} C_DIS
LIN {X 117.4858,Y -76.3648,Z 186,A -28.6155,B 2.898,C 0.2495,E1 3.0432,E2 481.8606} C_DIS
LIN {X 115.2481,Y -79.7027,Z 186,A -30.2714,B 2.8977,C 0.2536,E1 3.0406,E2 483.5197} C_DIS
LIN {X 111.3203,Y -85.1016,Z 186,A -32.7747,B 2.8973,C 0.2578,E1 3.0365,E2 485.9947} C_DIS
LIN {X 108.5569,Y -88.5997,Z 186,A -34.5306,B 2.897,C 0.2613,E1 3.0335,E2 487.7431} C_DIS
LIN {X 103.579,Y -94.3714,Z 186,A -37.3639,B 2.8966,C 0.2655,E1 3.0283,E2 490.5407} C_DIS
LIN {X 101.0554,Y -97.0692,Z 186,A -38.9505,B 2.8963,C 0.2694,E1 3.0252,E2 492.1389} C_DIS
LIN {X 97.9142,Y -100.2366,Z 186,A -40.8362,B 2.8959,C 0.2738,E1 3.0215,E2 494.0343} C_DIS
LIN {X 92.3545,Y -105.3813,Z 186,A -43.6848,B 2.8955,C 0.2777,E1 3.0157,E2 496.8517} C_DIS
LIN {X 89.1925,Y -108.0705,Z 186,A -45.9307,B 2.8947,C 0.2858,E1 3.0107,E2 499.1729} C_DIS
LIN {X 84.958,Y -111.4301,Z 186,A -47.7927,B 2.8947,C 0.2868,E1 3.0066,E2 500.9898} C_DIS
LIN {X 81.8782,Y -113.713,Z 186,A -48.9131,B 2.8947,C 0.2856,E1 3.0042,E2 502.0509} C_DIS
LIN {X 78.888,Y -115.8073,Z 186,A -50.4956,B 2.8944,C 0.289,E1 3.0006,E2 503.6467} C_DIS
LIN {X 72.241,Y -120.066,Z 186,A -53.5653,B 2.894,C 0.2928,E1 2.9934,E2 506.6974} C_DIS
LIN {X 68.628,Y -122.1666,Z 186,A -55.2829,B 2.8937,C 0.2955,E1 2.9892,E2 508.4174} C_DIS
LIN {X 64.7524,Y -124.2628,Z 186,A -57.0172,B 2.8935,C 0.2976,E1 2.9849,E2 510.1438} C_DIS
LIN {X 61.4867,Y -125.9111,Z 186,A -58.3999,B 2.8934,C 0.2987,E1 2.9815,E2 511.5121} C_DIS
LIN {X 59.0011,Y -127.0938,Z 186,A -59.9205,B 2.8929,C 0.3035,E1 2.9775,E2 513.0873} C_DIS
LIN {X 55.3571,Y -128.7229,Z 186,A -60.9323,B 2.8932,C 0.3004,E1 2.9751,E2 514.0158} C_DIS
LIN {X 52.6397,Y -129.8579,Z 186,A -62.3088,B 2.8929,C 0.3033,E1 2.9715,E2 515.4167} C_DIS
LIN {X 47.7942,Y -131.7184,Z 186,A -64.4332,B 2.8927,C 0.3058,E1 2.9659,E2 517.5429} C_DIS
LIN {X 44.1033,Y -132.9996,Z 186,A -65.9483,B 2.8925,C 0.3068,E1 2.962,E2 519.0477} C_DIS
LIN {X 40.86,Y -134.0315,Z 186,A -67.3065,B 2.8925,C 0.3079,E1 2.9583,E2 520.4023} C_DIS
LIN {X 37.2048,Y -135.0929,Z 186,A -68.9609,B 2.8922,C 0.3101,E1 2.9539,E2 522.071} C_DIS
LIN {X 32.5853,Y -136.2801,Z 186,A -70.82,B 2.8921,C 0.3111,E1 2.9488,E2 523.9189} C_DIS
LIN {X 28.1683,Y -137.2611,Z 186,A -73.0329,B 2.8916,C 0.3152,E1 2.9426,E2 526.1824} C_DIS
LIN {X 23.9445,Y -138.0624,Z 186,A -74.5244,B 2.8917,C 0.3144,E1 2.9386,E2 527.6386} C_DIS
LIN {X 18.7297,Y -138.8651,Z 186,A -76.5737,B 2.8917,C 0.3148,E1 2.933,E2 529.6744} C_DIS
LIN {X 14.744,Y -139.3439,Z 186,A -78.1656,B 2.8917,C 0.3152,E1 2.9286,E2 531.2604} C_DIS
LIN {X 10.3254,Y -139.7407,Z 186,A -79.9215,B 2.8917,C 0.3155,E1 2.9237,E2 533.0093} C_DIS
LIN {X 6.6542,Y -139.9641,Z 186,A -81.3631,B 2.8917,C 0.3155,E1 2.9197,E2 534.4432} C_DIS
LIN {X 2.9178,Y -140.0926,Z 186,A -82.9943,B 2.8915,C 0.3167,E1 2.9151,E2 536.0892} C_DIS
LIN {X 2.9178,Y -140.0926,Z 186,A -82.9943,B 2.8915,C 0.3167,E1 2.9151,E2 536.0892} C_DIS
Enddeposition()
LIN {X 1.0141,Y -141.0156,Z 186,A -83.2295,B 2.8053,C 0.3111,E1 2.8281,E2 536.3049} C_DIS
Startdeposition()
$VEL.CP = VEL_PRINT
LIN {X 3.8119,Y -140.9701,Z 186,A -81.8012,B 2.8056,C 0.3088,E1 2.8322,E2 534.8356} C_DIS
LIN {X 7.6231,Y -140.8164,Z 186,A -80.1781,B 2.8056,C 0.3078,E1 2.8368,E2 533.2015} C_DIS
LIN {X 11.7629,Y -140.53,Z 186,A -78.6122,B 2.8056,C 0.308,E1 2.8411,E2 531.6514} C_DIS
LIN {X 15.2573,Y -140.1937,Z 186,A -77.1574,B 2.8057,C 0.3071,E1 2.8452,E2 530.1919} C_DIS
LIN {X 21.7668,Y -139.3315,Z 186,A -74.3498,B 2.806,C 0.3046,E1 2.853,E2 527.3633} C_DIS
LIN {X 26.2381,Y -138.5591,Z 186,A -72.6651,B 2.806,C 0.3046,E1 2.8576,E2 525.6997} C_DIS
LIN {X 29.9914,Y -137.7954,Z 186,A -71.1551,B 2.8061,C 0.3037,E1 2.8617,E2 524.1952} C_DIS
LIN {X 33.8992,Y -136.8885,Z 186,A -69.4603,B 2.8063,C 0.3019,E1 2.8663,E2 522.4904} C_DIS
LIN {X 38.8678,Y -135.5613,Z 186,A -67.4127,B 2.8065,C 0.3003,E1 2.8718,E2 520.4473} C_DIS
LIN {X 42.6897,Y -134.4046,Z 186,A -65.9279,B 2.8065,C 0.2998,E1 2.8757,E2 518.9806} C_DIS
LIN {X 45.9613,Y -133.3213,Z 186,A -64.3733,B 2.8068,C 0.297,E1 2.8799,E2 517.4036} C_DIS
LIN {X 50.6635,Y -131.6068,Z 186,A -62.6374,B 2.8068,C 0.2971,E1 2.8844,E2 515.7078} C_DIS
LIN {X 53.9868,Y -130.2786,Z 186,A -61.0706,B 2.8071,C 0.2944,E1 2.8885,E2 514.1243} C_DIS
LIN {X 61.5532,Y -126.8812,Z 186,A -57.8088,B 2.8075,C 0.2909,E1 2.8967,E2 510.8753} C_DIS
LIN {X 65.4619,Y -124.9066,Z 186,A -56.1595,B 2.8076,C 0.2895,E1 2.9008,E2 509.2427} C_DIS
LIN {X 69.0619,Y -122.955,Z 186,A -54.421,B 2.8079,C 0.2863,E1 2.9051,E2 507.4927} C_DIS
LIN {X 71.8798,Y -121.3298,Z 186,A -53.2345,B 2.808,C 0.2854,E1 2.9079,E2 506.324} C_DIS
LIN {X 75.2991,Y -119.2369,Z 186,A -51.139,B 2.8087,C 0.2788,E1 2.913,E2 504.1623} C_DIS
LIN {X 79.0938,Y -116.7547,Z 186,A -49.7538,B 2.8087,C 0.2796,E1 2.9161,E2 502.8394} C_DIS
LIN {X 81.467,Y -115.1115,Z 186,A -48.0085,B 2.8093,C 0.2726,E1 2.9202,E2 501.0135} C_DIS
LIN {X 86.0732,Y -111.7097,Z 186,A -46.1398,B 2.8093,C 0.2724,E1 2.9242,E2 499.2069} C_DIS
LIN {X 88.7335,Y -109.6072,Z 186,A -44.6735,B 2.8096,C 0.269,E1 2.9274,E2 497.7272} C_DIS
LIN {X 92.015,Y -106.8678,Z 186,A -42.4965,B 2.8103,C 0.2617,E1 2.9322,E2 495.4874} C_DIS
LIN {X 97.318,Y -102.0623,Z 186,A -40.8609,B 2.8098,C 0.2673,E1 2.9352,E2 494.0261} C_DIS
LIN {X 101.558,Y -97.8446,Z 186,A -38.1748,B 2.8105,C 0.2599,E1 2.9405,E2 491.303} C_DIS
LIN {X 105.2383,Y -93.8746,Z 186,A -35.6459,B 2.8112,C 0.2521,E1 2.9453,E2 488.7268} C_DIS
LIN {X 108.3426,Y -90.2748,Z 186,A -34.19,B 2.8112,C 0.2522,E1 2.9479,E2 487.3351} C_DIS
LIN {X 111.1407,Y -86.8065,Z 186,A -32.5676,B 2.8114,C 0.2499,E1 2.9506,E2 485.737} C_DIS
LIN {X 114.579,Y -82.2143,Z 186,A -30.2144,B 2.8119,C 0.2442,E1 2.9545,E2 483.3789} C_DIS
LIN {X 116.7563,Y -79.0914,Z 186,A -28.6766,B 2.8122,C 0.2406,E1 2.957,E2 481.841} C_DIS
LIN {X 119.4674,Y -74.9344,Z 186,A -26.8248,B 2.8125,C 0.2373,E1 2.9597,E2 480.0103} C_DIS
LIN {X 121.7979,Y -71.0838,Z 186,A -25.2081,B 2.8127,C 0.2348,E1 2.962,E2 478.421} C_DIS
LIN {X 126.3349,Y -62.6618,Z 186,A -21.6243,B 2.8133,C 0.2279,E1 2.9667,E2 474.8757} C_DIS
LIN {X 128.9054,Y -57.1884,Z 186,A -19.0011,B 2.8139,C 0.2199,E1 2.9698,E2 472.2281} C_DIS
LIN {X 130.6183,Y -53.1602,Z 186,A -17.3466,B 2.8142,C 0.2164,E1 2.9715,E2 470.5891} C_DIS
LIN {X 131.8818,Y -49.944,Z 186,A -15.9504,B 2.8145,C 0.2128,E1 2.9729,E2 469.1929} C_DIS
LIN {X 133.9992,Y -43.9496,Z 186,A -13.1954,B 2.8151,C 0.2042,E1 2.9754,E2 466.4125} C_DIS
LIN {X 135.1861,Y -40.1493,Z 186,A -11.9759,B 2.8151,C 0.2036,E1 2.9764,E2 465.2459} C_DIS
LIN {X 136.4983,Y -35.435,Z 186,A -9.8936,B 2.8156,C 0.1973,E1 2.9779,E2 463.1493} C_DIS
LIN {X 137.2797,Y -32.2785,Z 186,A -8.8805,B 2.8156,C 0.1966,E1 2.9785,E2 462.177} C_DIS
LIN {X 138.4431,Y -26.8447,Z 186,A -6.6884,B 2.816,C 0.191,E1 2.9797,E2 459.992} C_DIS
LIN {X 139.0565,Y -23.4601,Z 186,A -5.4038,B 2.8162,C 0.1882,E1 2.9803,E2 458.7216} C_DIS
LIN {X 139.7319,Y -19.0408,Z 186,A -3.5665,B 2.8166,C 0.183,E1 2.9811,E2 456.8803} C_DIS
LIN {X 140.208,Y -15.125,Z 186,A -2.1722,B 2.8167,C 0.1805,E1 2.9815,E2 455.5127} C_DIS
LIN {X 140.5255,Y -11.8166,Z 186,A -0.8476,B 2.8169,C 0.1769,E1 2.9818,E2 454.1907} C_DIS
LIN {X 140.8125,Y -7.6994,Z 186,A 0.7987,B 2.8172,C 0.1725,E1 2.9821,E2 452.5474} C_DIS
LIN {X 140.9634,Y -4.0521,Z 186,A 2.1686,B 2.8174,C 0.1694,E1 2.9823,E2 451.1916} C_DIS
LIN {X 141.0249,Y 0.0534,Z 186,A 3.8956,B 2.8177,C 0.1642,E1 2.9823,E2 449.4557} C_DIS
LIN {X 140.9603,Y 4.1639,Z 186,A 5.3676,B 2.8179,C 0.1614,E1 2.9822,E2 448.009} C_DIS
LIN {X 140.7664,Y 8.4804,Z 186,A 7.0062,B 2.8181,C 0.1576,E1 2.982,E2 446.3849} C_DIS
LIN {X 140.5186,Y 11.8988,Z 186,A 8.3471,B 2.8183,C 0.1542,E1 2.9817,E2 445.05} C_DIS
LIN {X 140.1258,Y 15.8872,Z 186,A 9.9983,B 2.8185,C 0.1494,E1 2.9812,E2 443.3949} C_DIS
LIN {X 139.6315,Y 19.751,Z 186,A 11.3333,B 2.8186,C 0.1474,E1 2.9807,E2 442.0917} C_DIS
LIN {X 139.1665,Y 22.8004,Z 186,A 13.1116,B 2.8191,C 0.1388,E1 2.9799,E2 440.2431} C_DIS
LIN {X 138.2952,Y 27.5991,Z 186,A 15.2189,B 2.8194,C 0.1321,E1 2.9787,E2 438.118} C_DIS
LIN {X 136.9602,Y 33.6037,Z 186,A 16.8401,B 2.8194,C 0.1337,E1 2.9777,E2 436.6118} C_DIS
LIN {X 135.2038,Y 40.089,Z 186,A 19.5904,B 2.8197,C 0.1261,E1 2.9756,E2 433.8576} C_DIS
LIN {X 133.9739,Y 44.0256,Z 186,A 21.1284,B 2.8198,C 0.1229,E1 2.9743,E2 432.3369} C_DIS
LIN {X 132.7664,Y 47.5407,Z 186,A 22.5051,B 2.8199,C 0.1201,E1 2.9731,E2 430.977} C_DIS
LIN {X 131.631,Y 50.6013,Z 186,A 23.8476,B 2.8201,C 0.1164,E1 2.9717,E2 429.6319} C_DIS
LIN {X 130.1492,Y 54.2964,Z 186,A 25.3354,B 2.8202,C 0.1134,E1 2.9702,E2 428.1602} C_DIS
LIN {X 128.7242,Y 57.5934,Z 186,A 26.6808,B 2.8203,C 0.1107,E1 2.9687,E2 426.8291} C_DIS
LIN {X 127.3135,Y 60.6481,Z 186,A 28.0056,B 2.8204,C 0.1076,E1 2.9671,E2 425.5093} C_DIS
LIN {X 125.9451,Y 63.4436,Z 186,A 29.2744,B 2.8206,C 0.1043,E1 2.9655,E2 424.2395} C_DIS
LIN {X 124.0489,Y 67.0784,Z 186,A 30.907,B 2.8206,C 0.1004,E1 2.9634,E2 422.6107} C_DIS
LIN {X 121.8984,Y 70.9109,Z 186,A 32.6142,B 2.8208,C 0.0967,E1 2.961,E2 420.913} C_DIS
LIN {X 119.5047,Y 74.8753,Z 186,A 34.4445,B 2.821,C 0.0926,E1 2.9584,E2 419.0889} C_DIS
LIN {X 116.9608,Y 78.7893,Z 186,A 36.2374,B 2.821,C 0.089,E1 2.9556,E2 417.3088} C_DIS
LIN {X 114.3927,Y 82.4737,Z 186,A 38.0115,B 2.8212,C 0.0852,E1 2.9528,E2 415.5408} C_DIS
LIN {X 111.962,Y 85.7438,Z 186,A 39.849,B 2.8214,C 0.0798,E1 2.9496,E2 413.6793} C_DIS
LIN {X 109.5655,Y 88.7861,Z 186,A 41.0864,B 2.8214,C 0.0793,E1 2.9475,E2 412.485} C_DIS
LIN {X 106.6747,Y 92.2392,Z 186,A 42.8554,B 2.8214,C 0.0758,E1 2.9443,E2 410.7234} C_DIS
LIN {X 103.6676,Y 95.6063,Z 186,A 44.6154,B 2.8216,C 0.0725,E1 2.941,E2 408.9726} C_DIS
LIN {X 100.4642,Y 98.9672,Z 186,A 46.438,B 2.8216,C 0.0691,E1 2.9375,E2 407.158} C_DIS
LIN {X 97.2339,Y 102.1427,Z 186,A 48.5842,B 2.8218,C 0.0628,E1 2.9331,E2 404.9723} C_DIS
LIN {X 93.9944,Y 105.1311,Z 186,A 49.9214,B 2.8218,C 0.0632,E1 2.9304,E2 403.6931} C_DIS
LIN {X 90.4798,Y 108.1708,Z 186,A 51.8504,B 2.8218,C 0.0592,E1 2.9263,E2 401.7587} C_DIS
LIN {X 86.5813,Y 111.3158,Z 186,A 53.7304,B 2.8219,C 0.0568,E1 2.9222,E2 399.8985} C_DIS
LIN {X 83.1078,Y 113.9331,Z 186,A 55.677,B 2.8219,C 0.0522,E1 2.9178,E2 397.9288} C_DIS
LIN {X 80.2011,Y 115.9975,Z 186,A 56.8494,B 2.822,C 0.052,E1 2.9152,E2 396.7917} C_DIS
LIN {X 76.4291,Y 118.5169,Z 186,A 58.6543,B 2.822,C 0.0493,E1 2.911,E2 394.9917} C_DIS
LIN {X 72.7968,Y 120.7814,Z 186,A 60.3244,B 2.822,C 0.0472,E1 2.907,E2 393.3304} C_DIS
LIN {X 68.8756,Y 123.0598,Z 186,A 62.1393,B 2.8221,C 0.0446,E1 2.9026,E2 391.519} C_DIS
LIN {X 65.7739,Y 124.7428,Z 186,A 63.7923,B 2.8221,C 0.0409,E1 2.8985,E2 389.8382} C_DIS
LIN {X 62.4358,Y 126.4463,Z 186,A 64.8764,B 2.8221,C 0.0422,E1 2.8959,E2 388.81} C_DIS
LIN {X 59.4751,Y 127.8661,Z 186,A 66.2413,B 2.8221,C 0.0402,E1 2.8924,E2 387.4414} C_DIS
LIN {X 56.3831,Y 129.2597,Z 186,A 67.4477,B 2.8222,C 0.0398,E1 2.8894,E2 386.2568} C_DIS
LIN {X 53.0502,Y 130.6626,Z 186,A 68.9801,B 2.8222,C 0.0376,E1 2.8854,E2 384.7167} C_DIS
LIN {X 49.929,Y 131.8874,Z 186,A 70.3719,B 2.8222,C 0.0358,E1 2.8818,E2 383.3213} C_DIS
LIN {X 46.6717,Y 133.075,Z 186,A 72.0803,B 2.8222,C 0.0321,E1 2.8772,E2 381.5753} C_DIS
LIN {X 43.1904,Y 134.2446,Z 186,A 73.6514,B 2.8223,C 0.0301,E1 2.873,E2 379.9945} C_DIS
LIN {X 38.9884,Y 135.526,Z 186,A 75.0863,B 2.8223,C 0.031,E1 2.8693,E2 378.6044} C_DIS
LIN {X 36.1232,Y 136.3163,Z 186,A 76.3684,B 2.8223,C 0.0294,E1 2.8658,E2 377.3131} C_DIS
LIN {X 31.9928,Y 137.3456,Z 186,A 77.9646,B 2.8223,C 0.029,E1 2.8615,E2 375.7343} C_DIS
LIN {X 28.0809,Y 138.1972,Z 186,A 79.4665,B 2.8223,C 0.0287,E1 2.8574,E2 374.2485} C_DIS
LIN {X 24.0266,Y 138.9619,Z 186,A 81.0938,B 2.8223,C 0.028,E1 2.8529,E2 372.628} C_DIS
LIN {X 19.2483,Y 139.7033,Z 186,A 83.1415,B 2.8223,C 0.0264,E1 2.8473,E2 370.5704} C_DIS
LIN {X 15.2985,Y 140.1893,Z 186,A 84.6904,B 2.8223,C 0.0261,E1 2.843,E2 369.0306} C_DIS
LIN {X 11.5632,Y 140.5469,Z 186,A 86.2196,B 2.8223,C 0.0255,E1 2.8387,E2 367.5013} C_DIS
LIN {X 7.2954,Y 140.8328,Z 186,A 87.8863,B 2.8223,C 0.0254,E1 2.8341,E2 365.8443} C_DIS
LIN {X 3.8919,Y 140.9678,Z 186,A 89.3023,B 2.8223,C 0.0249,E1 2.8301,E2 364.4247} C_DIS
LIN {X -0.3714,Y 141.0217,Z 186,A 91.0541,B 2.8223,C 0.0245,E1 2.8252,E2 362.6713} C_DIS
LIN {X -4.5882,Y 140.9485,Z 186,A 92.8063,B 2.8223,C 0.0241,E1 2.8203,E2 360.915} C_DIS
LIN {X -12.1094,Y 140.5008,Z 186,A 95.7986,B 2.8223,C 0.0247,E1 2.812,E2 357.9328} C_DIS
LIN {X -16.0917,Y 140.1016,Z 186,A 97.4788,B 2.8223,C 0.0247,E1 2.8073,E2 356.2466} C_DIS
LIN {X -19.9226,Y 139.607,Z 186,A 99.3916,B 2.8223,C 0.023,E1 2.8019,E2 354.2915} C_DIS
LIN {X -23.9635,Y 138.9725,Z 186,A 100.8811,B 2.8223,C 0.0246,E1 2.7978,E2 352.8245} C_DIS
LIN {X -32.5708,Y 137.2092,Z 186,A 104.1231,B 2.8223,C 0.0281,E1 2.7891,E2 349.6257} C_DIS
LIN {X -34.77,Y 136.6676,Z 186,A 105.5921,B 2.8223,C 0.0255,E1 2.7849,E2 348.0883} C_DIS
LIN {X -38.6954,Y 135.6104,Z 186,A 106.981,B 2.8223,C 0.028,E1 2.7813,E2 346.7335} C_DIS
LIN {X -42.5239,Y 134.4576,Z 186,A 108.4697,B 2.8223,C 0.0299,E1 2.7773,E2 345.2627} C_DIS
LIN {X -45.8913,Y 133.3455,Z 186,A 110.2007,B 2.8223,C 0.0295,E1 2.7727,E2 343.4961} C_DIS
LIN {X -51.8318,Y 131.1527,Z 186,A 112.9122,B 2.8223,C 0.0311,E1 2.7655,E2 340.7689} C_DIS
LIN {X -55.117,Y 129.8066,Z 186,A 114.1959,B 2.8223,C 0.0333,E1 2.7623,E2 339.506} C_DIS
LIN {X -58.5771,Y 128.2813,Z 186,A 116.3022,B 2.8223,C 0.032,E1 2.7568,E2 337.3286} C_DIS
LIN {X -63.4732,Y 125.93,Z 186,A 117.9428,B 2.8223,C 0.0374,E1 2.7528,E2 335.7611} C_DIS
LIN {X -67.1199,Y 124.0266,Z 186,A 119.6974,B 2.8223,C 0.039,E1 2.7485,E2 333.9972} C_DIS
LIN {X -70.1552,Y 122.3349,Z 186,A 121.7619,B 2.8223,C 0.0377,E1 2.7433,E2 331.851} C_DIS
LIN {X -75.0562,Y 119.3906,Z 186,A 123.4687,B 2.8221,C 0.0438,E1 2.7394,E2 330.2239} C_DIS
LIN {X -79.4713,Y 116.4987,Z 186,A 125.7255,B 2.8221,C 0.0465,E1 2.7341,E2 327.9545} C_DIS
LIN {X -81.9961,Y 114.735,Z 186,A 127.2246,B 2.8221,C 0.0473,E1 2.7307,E2 326.425} C_DIS
LIN {X -84.8292,Y 112.6566,Z 186,A 128.4592,B 2.8221,C 0.0504,E1 2.7279,E2 325.2158} C_DIS
LIN {X -88.3089,Y 109.9505,Z 186,A 130.3331,B 2.822,C 0.053,E1 2.7238,E2 323.3327} C_DIS
LIN {X -91.8298,Y 107.0273,Z 186,A 132.1946,B 2.822,C 0.0563,E1 2.7198,E2 321.4723} C_DIS
LIN {X -95.7934,Y 103.4953,Z 186,A 134.4911,B 2.8219,C 0.0596,E1 2.7151,E2 319.1597} C_DIS
LIN {X -99.1087,Y 100.325,Z 186,A 136.3419,B 2.8218,C 0.0632,E1 2.7114,E2 317.3119} C_DIS
LIN {X -102.1871,Y 97.1874,Z 186,A 138.2257,B 2.8218,C 0.0663,E1 2.7077,E2 315.417} C_DIS
LIN {X -106.6707,Y 92.2438,Z 186,A 141.0849,B 2.8216,C 0.0712,E1 2.7023,E2 312.5411} C_DIS
LIN {X -108.8051,Y 89.7163,Z 186,A 142.5442,B 2.8216,C 0.0736,E1 2.6997,E2 311.0681} C_DIS
LIN {X -111.8113,Y 85.9408,Z 186,A 144.493,B 2.8214,C 0.0779,E1 2.6964,E2 309.1224} C_DIS
LIN {X -114.5009,Y 82.3235,Z 186,A 146.3684,B 2.8213,C 0.0818,E1 2.6933,E2 307.2427} C_DIS
LIN {X -118.7226,Y 76.108,Z 186,A 149.5616,B 2.8211,C 0.0883,E1 2.6883,E2 304.034} C_DIS
LIN {X -120.9365,Y 72.5397,Z 186,A 151.4038,B 2.821,C 0.0919,E1 2.6856,E2 302.1757} C_DIS
LIN {X -123.1428,Y 68.7278,Z 186,A 153.3618,B 2.8209,C 0.0956,E1 2.6829,E2 300.1974} C_DIS
LIN {X -125.4528,Y 64.4106,Z 186,A 155.2664,B 2.8207,C 0.1008,E1 2.6804,E2 298.3051} C_DIS
LIN {X -127.1032,Y 61.0885,Z 186,A 156.6971,B 2.8205,C 0.1049,E1 2.6787,E2 296.8853} C_DIS
LIN {X -128.4408,Y 58.2269,Z 186,A 158.2407,B 2.8205,C 0.1072,E1 2.6768,E2 295.3093} C_DIS
LIN {X -130.0232,Y 54.5983,Z 186,A 159.8363,B 2.8203,C 0.1114,E1 2.6751,E2 293.7165} C_DIS
LIN {X -131.2896,Y 51.4796,Z 186,A 161.2629,B 2.8201,C 0.1147,E1 2.6736,E2 292.2833} C_DIS
LIN {X -132.4712,Y 48.3594,Z 186,A 162.7765,B 2.8201,C 0.1178,E1 2.6721,E2 290.7503} C_DIS
LIN {X -133.7191,Y 44.7909,Z 186,A 164.327,B 2.8199,C 0.1218,E1 2.6707,E2 289.199} C_DIS
LIN {X -134.8101,Y 41.3911,Z 186,A 165.7059,B 2.8197,C 0.1259,E1 2.6695,E2 287.8304} C_DIS
LIN {X -135.7549,Y 38.1788,Z 186,A 167.236,B 2.8195,C 0.129,E1 2.6683,E2 286.2794} C_DIS
LIN {X -136.6219,Y 34.95,Z 186,A 168.7081,B 2.8194,C 0.1323,E1 2.6673,E2 284.7934} C_DIS
LIN {X -137.4243,Y 31.648,Z 186,A 170.2664,B 2.8192,C 0.1355,E1 2.6663,E2 283.2131} C_DIS
LIN {X -138.602,Y 26.0137,Z 186,A 172.72,B 2.8189,C 0.1416,E1 2.6649,E2 280.7461} C_DIS
LIN {X -139.7861,Y 18.6273,Z 186,A 175.741,B 2.8185,C 0.1501,E1 2.6637,E2 277.7297} C_DIS
LIN {X -140.1901,Y 15.291,Z 186,A 177.2798,B 2.8183,C 0.1533,E1 2.6632,E2 276.1692} C_DIS
LIN {X -140.5419,Y 11.6227,Z 186,A 178.8554,B 2.8181,C 0.1573,E1 2.6628,E2 274.5843} C_DIS
LIN {X -140.9386,Y 4.8697,Z 186,A -177.965,B 2.8177,C 0.1636,E1 2.6623,E2 271.3497} C_DIS
LIN {X -141.016,Y 1.4318,Z 186,A -176.7865,B 2.8175,C 0.1682,E1 2.6623,E2 270.2011} C_DIS
LIN {X -140.9913,Y -2.9936,Z 186,A -174.8602,B 2.8172,C 0.1729,E1 2.6623,E2 268.2589} C_DIS
LIN {X -140.8966,Y -5.9509,Z 186,A -173.0907,B 2.8171,C 0.1743,E1 2.6626,E2 266.4148} C_DIS
LIN {X -140.6242,Y -10.5819,Z 186,A -171.7451,B 2.8166,C 0.1815,E1 2.6628,E2 265.1421} C_DIS
LIN {X -139.7464,Y -18.9298,Z 186,A -168.2177,B 2.816,C 0.1906,E1 2.6639,E2 261.6015} C_DIS
LIN {X -138.6889,Y -25.5519,Z 186,A -165.1035,B 2.8156,C 0.1968,E1 2.6654,E2 258.4372} C_DIS
LIN {X -137.8937,Y -29.5362,Z 186,A -163.4027,B 2.8153,C 0.2011,E1 2.6663,E2 256.7306} C_DIS
LIN {X -137.0596,Y -33.1914,Z 186,A -161.8594,B 2.815,C 0.2052,E1 2.6673,E2 255.1854} C_DIS
LIN {X -136.176,Y -36.6493,Z 186,A -160.2953,B 2.8148,C 0.2087,E1 2.6684,E2 253.6068} C_DIS
LIN {X -134.9682,Y -40.8743,Z 186,A -158.4264,B 2.8144,C 0.2132,E1 2.6699,E2 251.7276} C_DIS
LIN {X -133.8306,Y -44.4559,Z 186,A -156.8274,B 2.8141,C 0.217,E1 2.6713,E2 250.1196} C_DIS
LIN {X -131.7192,Y -50.3744,Z 186,A -154.1049,B 2.8137,C 0.2231,E1 2.6739,E2 247.3756} C_DIS
LIN {X -130.3548,Y -53.8042,Z 186,A -152.553,B 2.8134,C 0.2267,E1 2.6756,E2 245.8173} C_DIS
LIN {X -129.2963,Y -56.2984,Z 186,A -151.3483,B 2.8132,C 0.2291,E1 2.6769,E2 244.5989} C_DIS
LIN {X -127.437,Y -60.3898,Z 186,A -149.4991,B 2.8128,C 0.2336,E1 2.6791,E2 242.7473} C_DIS
LIN {X -125.8053,Y -63.7183,Z 186,A -147.96,B 2.8125,C 0.2372,E1 2.681,E2 241.2044} C_DIS
LIN {X -124.5375,Y -66.1647,Z 186,A -146.3667,B 2.8125,C 0.2381,E1 2.6832,E2 239.5472} C_DIS
LIN {X -122.5957,Y -69.698,Z 186,A -144.9726,B 2.812,C 0.243,E1 2.6851,E2 238.1869} C_DIS
LIN {X -120.2893,Y -73.607,Z 186,A -143.0972,B 2.8116,C 0.2472,E1 2.6878,E2 236.3078} C_DIS
LIN {X -117.8724,Y -77.4183,Z 186,A -141.1324,B 2.8113,C 0.2509,E1 2.6908,E2 234.3257} C_DIS
LIN {X -115.2403,Y -81.2845,Z 186,A -139.2781,B 2.8109,C 0.2553,E1 2.6937,E2 232.4782} C_DIS
LIN {X -109.2629,Y -89.1578,Z 186,A -135.0636,B 2.8102,C 0.2632,E1 2.701,E2 228.238} C_DIS
LIN {X -105.2991,Y -93.8068,Z 186,A -132.3704,B 2.8098,C 0.2673,E1 2.7059,E2 225.5164} C_DIS
LIN {X -102.7227,Y -96.6208,Z 186,A -130.7833,B 2.8095,C 0.2702,E1 2.709,E2 223.9245} C_DIS
LIN {X -99.6897,Y -99.7478,Z 186,A -128.123,B 2.8096,C 0.2694,E1 2.7145,E2 221.1414} C_DIS
LIN {X -94.7853,Y -104.4185,Z 186,A -126.3082,B 2.8087,C 0.2788,E1 2.7179,E2 219.4566} C_DIS
LIN {X -91.0965,Y -107.6522,Z 186,A -124.0592,B 2.8085,C 0.281,E1 2.7228,E2 217.1725} C_DIS
LIN {X -87.5995,Y -110.5165,Z 186,A -122.1795,B 2.8082,C 0.2838,E1 2.7269,E2 215.287} C_DIS
LIN {X -81.9424,Y -114.7734,Z 186,A -119.2361,B 2.8078,C 0.2879,E1 2.7335,E2 212.3345} C_DIS
LIN {X -78.1471,Y -117.3906,Z 186,A -117.2824,B 2.8075,C 0.2902,E1 2.738,E2 210.3696} C_DIS
LIN {X -74.0842,Y -119.9966,Z 186,A -115.2544,B 2.8073,C 0.2925,E1 2.7429,E2 208.3322} C_DIS
LIN {X -70.3339,Y -122.2324,Z 186,A -113.4428,B 2.8071,C 0.2946,E1 2.7472,E2 206.5152} C_DIS
LIN {X -64.6801,Y -125.3157,Z 186,A -110.7425,B 2.8068,C 0.2972,E1 2.7539,E2 203.803} C_DIS
LIN {X -61.0361,Y -127.1282,Z 186,A -109.2193,B 2.8065,C 0.2997,E1 2.7577,E2 202.2977} C_DIS
LIN {X -58.2758,Y -128.4189,Z 186,A -107.765,B 2.8065,C 0.2997,E1 2.7615,E2 200.8132} C_DIS
LIN {X -54.3597,Y -130.1228,Z 186,A -106.1742,B 2.8063,C 0.3022,E1 2.7655,E2 199.2421} C_DIS
LIN {X -51.2535,Y -131.3775,Z 186,A -104.8743,B 2.8061,C 0.3038,E1 2.7689,E2 197.9504} C_DIS
LIN {X -48.578,Y -132.3922,Z 186,A -103.3878,B 2.8062,C 0.3028,E1 2.7729,E2 196.4187} C_DIS
LIN {X -42.0136,Y -134.6195,Z 186,A -100.635,B 2.8059,C 0.3052,E1 2.7802,E2 193.6741} C_DIS
LIN {X -37.1592,Y -136.0394,Z 186,A -98.6961,B 2.8057,C 0.3071,E1 2.7854,E2 191.7508} C_DIS
LIN {X -33.7063,Y -136.9355,Z 186,A -97.2638,B 2.8057,C 0.308,E1 2.7892,E2 190.3204} C_DIS
LIN {X -30.1823,Y -137.7541,Z 186,A -95.6779,B 2.8057,C 0.3079,E1 2.7936,E2 188.7178} C_DIS
LIN {X -26.9437,Y -138.4242,Z 186,A -94.4268,B 2.8055,C 0.309,E1 2.797,E2 187.4792} C_DIS
LIN {X -23.4345,Y -139.0607,Z 186,A -92.8921,B 2.8055,C 0.3089,E1 2.8013,E2 185.932} C_DIS
LIN {X -19.88,Y -139.6131,Z 186,A -91.4382,B 2.8055,C 0.3093,E1 2.8053,E2 184.4786} C_DIS
LIN {X -15.661,Y -140.1503,Z 186,A -89.6118,B 2.8055,C 0.3089,E1 2.8104,E2 182.6379} C_DIS
LIN {X -11.8915,Y -140.5192,Z 186,A -88.1976,B 2.8055,C 0.3098,E1 2.8143,E2 181.2405} C_DIS
LIN {X -8.1235,Y -140.7884,Z 186,A -86.5213,B 2.8055,C 0.3089,E1 2.819,E2 179.5438} C_DIS
LIN {X -3.8667,Y -140.9685,Z 186,A -84.9146,B 2.8055,C 0.3096,E1 2.8235,E2 177.9536} C_DIS
LIN {X -0.0298,Y -141.0236,Z 186,A -83.2776,B 2.8055,C 0.3088,E1 2.8281,E2 176.305} C_DIS
LIN {X -0.0298,Y -141.0236,Z 186,A -83.2776,B 2.8055,C 0.3088,E1 2.8281,E2 176.305} C_DIS
Enddeposition()
LIN {X 1.0204,Y -141.9169,Z 186,A -83.2329,B 2.8043,C 0.3128,E1 2.8271,E2 176.3437} C_DIS
Startdeposition()
$VEL.CP = VEL_PRINT
LIN {X -1.5487,Y -141.915,Z 186,A -84.6815,B 2.8039,C 0.3159,E1 2.8229,E2 177.8502} C_DIS
LIN {X -5.8209,Y -141.8023,Z 186,A -86.3076,B 2.8039,C 0.3153,E1 2.8184,E2 179.4633} C_DIS
LIN {X -10.1303,Y -141.5595,Z 186,A -88.083,B 2.8039,C 0.3156,E1 2.8135,E2 181.2441} C_DIS
LIN {X -13.6831,Y -141.2602,Z 186,A -89.4649,B 2.804,C 0.3151,E1 2.8096,E2 182.6185} C_DIS
LIN {X -17.3045,Y -140.8632,Z 186,A -90.9406,B 2.804,C 0.3149,E1 2.8055,E2 184.0955} C_DIS
LIN {X -21.1942,Y -140.3307,Z 186,A -92.6077,B 2.804,C 0.3151,E1 2.8009,E2 185.7747} C_DIS
LIN {X -24.9192,Y -139.7163,Z 186,A -94.133,B 2.804,C 0.3146,E1 2.7967,E2 187.3006} C_DIS
LIN {X -28.3973,Y -139.0511,Z 186,A -95.5271,B 2.8041,C 0.3139,E1 2.7929,E2 188.6903} C_DIS
LIN {X -32.4199,Y -138.1709,Z 186,A -97.1642,B 2.8042,C 0.313,E1 2.7884,E2 190.3245} C_DIS
LIN {X -35.702,Y -137.3594,Z 186,A -98.6554,B 2.8042,C 0.313,E1 2.7843,E2 191.8336} C_DIS
LIN {X -40.734,Y -135.9522,Z 186,A -101.5239,B 2.8039,C 0.3163,E1 2.7763,E2 194.8074} C_DIS
LIN {X -46.6822,Y -134.0237,Z 186,A -103.6747,B 2.8043,C 0.3122,E1 2.7708,E2 196.9074} C_DIS
LIN {X -50.6639,Y -132.5721,Z 186,A -104.9684,B 2.8047,C 0.3084,E1 2.7675,E2 198.1438} C_DIS
LIN {X -53.7036,Y -131.3695,Z 186,A -106.3255,B 2.8049,C 0.3074,E1 2.764,E2 199.5064} C_DIS
LIN {X -56.8497,Y -130.0384,Z 186,A -107.7259,B 2.8049,C 0.3063,E1 2.7604,E2 200.9099} C_DIS
LIN {X -59.9013,Y -128.6604,Z 186,A -109.1115,B 2.8051,C 0.3051,E1 2.7569,E2 202.3004} C_DIS
LIN {X -63.1564,Y -127.0943,Z 186,A -110.6266,B 2.8052,C 0.3038,E1 2.753,E2 203.8235} C_DIS
LIN {X -67.2148,Y -124.9971,Z 186,A -112.6401,B 2.8054,C 0.3026,E1 2.748,E2 205.8607} C_DIS
LIN {X -71.5556,Y -122.5644,Z 186,A -114.6075,B 2.8057,C 0.2999,E1 2.7432,E2 207.8225} C_DIS
LIN {X -75.2429,Y -120.3358,Z 186,A -116.4087,B 2.8059,C 0.2979,E1 2.7389,E2 209.6323} C_DIS
LIN {X -79.0753,Y -117.8529,Z 186,A -118.2997,B 2.8061,C 0.2955,E1 2.7345,E2 211.5299} C_DIS
LIN {X -82.5264,Y -115.4621,Z 186,A -120.0372,B 2.8064,C 0.2932,E1 2.7305,E2 213.2733} C_DIS
LIN {X -86.4763,Y -112.5346,Z 186,A -122.041,B 2.8067,C 0.2902,E1 2.726,E2 215.2797} C_DIS
LIN {X -89.6969,Y -109.9844,Z 186,A -123.8007,B 2.8069,C 0.288,E1 2.7222,E2 217.0531} C_DIS
LIN {X -93.1907,Y -107.0402,Z 186,A -125.5074,B 2.8073,C 0.2841,E1 2.7186,E2 218.7408} C_DIS
LIN {X -95.8174,Y -104.6958,Z 186,A -127.1968,B 2.8074,C 0.2829,E1 2.715,E2 220.4668} C_DIS
LIN {X -100.0309,Y -100.6772,Z 186,A -129.3374,B 2.808,C 0.2776,E1 2.7107,E2 222.5784} C_DIS
LIN {X -102.1632,Y -98.5132,Z 186,A -130.8606,B 2.808,C 0.2766,E1 2.7077,E2 224.142} C_DIS
LIN {X -104.8635,Y -95.634,Z 186,A -132.5513,B 2.8083,C 0.2739,E1 2.7045,E2 225.8458} C_DIS
LIN {X -108.3254,Y -91.694,Z 186,A -134.71,B 2.8087,C 0.2697,E1 2.7005,E2 228.0097} C_DIS
LIN {X -111.2217,Y -88.1585,Z 186,A -136.6093,B 2.8091,C 0.2661,E1 2.6972,E2 229.9159} C_DIS
LIN {X -115.0167,Y -83.1462,Z 186,A -139.0455,B 2.8096,C 0.2601,E1 2.6931,E2 232.3376} C_DIS
LIN {X -116.9644,Y -80.383,Z 186,A -140.7184,B 2.8098,C 0.2583,E1 2.6904,E2 234.052} C_DIS
LIN {X -119.6499,Y -76.3286,Z 186,A -142.73,B 2.8102,C 0.254,E1 2.6873,E2 236.0696} C_DIS
LIN {X -121.9871,Y -72.5346,Z 186,A -144.6013,B 2.8105,C 0.2501,E1 2.6846,E2 237.95} C_DIS
LIN {X -124.2342,Y -68.6147,Z 186,A -146.6251,B 2.8109,C 0.2465,E1 2.6818,E2 240.0002} C_DIS
LIN {X -126.6319,Y -64.078,Z 186,A -148.6092,B 2.8113,C 0.2411,E1 2.6792,E2 241.9717} C_DIS
LIN {X -128.273,Y -60.7272,Z 186,A -150.2329,B 2.8116,C 0.2378,E1 2.6772,E2 243.6106} C_DIS
LIN {X -130.2403,Y -56.3825,Z 186,A -152.2481,B 2.812,C 0.2333,E1 2.6749,E2 245.6372} C_DIS
LIN {X -131.9517,Y -52.2591,Z 186,A -154.0973,B 2.8124,C 0.2288,E1 2.673,E2 247.4919} C_DIS
LIN {X -133.2968,Y -48.7226,Z 186,A -155.8805,B 2.8126,C 0.2257,E1 2.6712,E2 249.3086} C_DIS
LIN {X -134.7215,Y -44.6287,Z 186,A -157.5364,B 2.813,C 0.2208,E1 2.6697,E2 250.951} C_DIS
LIN {X -135.8399,Y -41.101,Z 186,A -159.0894,B 2.8133,C 0.217,E1 2.6684,E2 252.5113} C_DIS
LIN {X -136.7275,Y -38.0419,Z 186,A -160.4594,B 2.8135,C 0.2139,E1 2.6674,E2 253.8919} C_DIS
LIN {X -137.6889,Y -34.4037,Z 186,A -162.0183,B 2.8138,C 0.2099,E1 2.6663,E2 255.4552} C_DIS
LIN {X -138.4192,Y -31.3337,Z 186,A -163.4281,B 2.814,C 0.2069,E1 2.6654,E2 256.8825} C_DIS
LIN {X -139.6328,Y -25.3858,Z 186,A -165.7899,B 2.8146,C 0.1999,E1 2.6641,E2 259.2311} C_DIS
LIN {X -140.2523,Y -21.7003,Z 186,A -167.5607,B 2.8148,C 0.1966,E1 2.6633,E2 261.0358} C_DIS
LIN {X -140.7386,Y -18.2843,Z 186,A -169.0915,B 2.815,C 0.1932,E1 2.6627,E2 262.5841} C_DIS
LIN {X -141.411,Y -12.0246,Z 186,A -171.405,B 2.8155,C 0.1853,E1 2.6621,E2 264.866} C_DIS
LIN {X -141.593,Y -9.6702,Z 186,A -172.9118,B 2.8156,C 0.1845,E1 2.6617,E2 266.4454} C_DIS
LIN {X -141.817,Y -5.444,Z 186,A -174.5622,B 2.8159,C 0.1795,E1 2.6615,E2 268.087} C_DIS
LIN {X -141.9205,Y -0.7438,Z 186,A -176.5189,B 2.8162,C 0.1743,E1 2.6615,E2 270.0502} C_DIS
LIN {X -141.8803,Y 3.4499,Z 186,A -178.4399,B 2.8165,C 0.1703,E1 2.6615,E2 272} C_DIS
LIN {X -141.6767,Y 8.3379,Z 186,A 179.5463,B 2.8168,C 0.1649,E1 2.6618,E2 274.0176} C_DIS
LIN {X -141.4059,Y 12.0849,Z 186,A 178.0087,B 2.8171,C 0.1607,E1 2.6622,E2 275.5568} C_DIS
LIN {X -141.0152,Y 16.0288,Z 186,A 176.3803,B 2.8173,C 0.1563,E1 2.6626,E2 277.188} C_DIS
LIN {X -140.6875,Y 18.6738,Z 186,A 175.1805,B 2.8174,C 0.1537,E1 2.6631,E2 278.403} C_DIS
LIN {X -139.8864,Y 23.9537,Z 186,A 172.9931,B 2.8178,C 0.1479,E1 2.664,E2 280.5931} C_DIS
LIN {X -138.3876,Y 31.4721,Z 186,A 169.9609,B 2.8182,C 0.1391,E1 2.6657,E2 283.6151} C_DIS
LIN {X -137.7933,Y 33.9876,Z 186,A 168.5951,B 2.8182,C 0.1373,E1 2.6666,E2 285.022} C_DIS
LIN {X -136.8332,Y 37.6642,Z 186,A 166.8853,B 2.8185,C 0.1338,E1 2.6679,E2 286.7535} C_DIS
LIN {X -135.7404,Y 41.4262,Z 186,A 165.325,B 2.8187,C 0.1294,E1 2.6691,E2 288.3098} C_DIS
LIN {X -134.5991,Y 44.9964,Z 186,A 163.7532,B 2.8188,C 0.1256,E1 2.6705,E2 289.8881} C_DIS
LIN {X -133.4342,Y 48.3416,Z 186,A 162.2407,B 2.819,C 0.1221,E1 2.6719,E2 291.4101} C_DIS
LIN {X -132.1458,Y 51.7607,Z 186,A 160.6348,B 2.8191,C 0.1187,E1 2.6735,E2 293.0318} C_DIS
LIN {X -130.8283,Y 55.0054,Z 186,A 159.1817,B 2.8193,C 0.1152,E1 2.6751,E2 294.4889} C_DIS
LIN {X -129.3666,Y 58.361,Z 186,A 157.639,B 2.8194,C 0.1116,E1 2.6768,E2 296.0388} C_DIS
LIN {X -127.8093,Y 61.6979,Z 186,A 156.0854,B 2.8196,C 0.1081,E1 2.6787,E2 297.5999} C_DIS
LIN {X -126.2103,Y 64.9062,Z 186,A 154.5174,B 2.8196,C 0.1049,E1 2.6807,E2 299.1822} C_DIS
LIN {X -124.2282,Y 68.6256,Z 186,A 152.6695,B 2.8198,C 0.1013,E1 2.6832,E2 301.0476} C_DIS
LIN {X -121.9434,Y 72.6079,Z 186,A 150.7487,B 2.82,C 0.0971,E1 2.6859,E2 302.9756} C_DIS
LIN {X -119.5714,Y 76.4511,Z 186,A 148.8546,B 2.8201,C 0.0931,E1 2.6887,E2 304.8773} C_DIS
LIN {X -116.5875,Y 80.9288,Z 186,A 146.5609,B 2.8202,C 0.0885,E1 2.6923,E2 307.1847} C_DIS
LIN {X -114.5376,Y 83.805,Z 186,A 145.0481,B 2.8203,C 0.0857,E1 2.6948,E2 308.7074} C_DIS
LIN {X -111.6359,Y 87.6328,Z 186,A 143.0637,B 2.8205,C 0.0816,E1 2.6982,E2 310.6962} C_DIS
LIN {X -109.1879,Y 90.6649,Z 186,A 141.4494,B 2.8205,C 0.0784,E1 2.7011,E2 312.3145} C_DIS
LIN {X -106.1925,Y 94.1556,Z 186,A 139.4219,B 2.8206,C 0.0753,E1 2.7048,E2 314.3621} C_DIS
LIN {X -103.4978,Y 97.1104,Z 186,A 137.8256,B 2.8207,C 0.072,E1 2.7079,E2 315.9549} C_DIS
LIN {X -100.3427,Y 100.3674,Z 186,A 135.9617,B 2.8208,C 0.0685,E1 2.7115,E2 317.8216} C_DIS
LIN {X -97.3103,Y 103.3093,Z 186,A 134.1772,B 2.8208,C 0.0657,E1 2.7151,E2 319.6148} C_DIS
LIN {X -93.9899,Y 106.339,Z 186,A 132.493,B 2.821,C 0.0618,E1 2.7186,E2 321.2812} C_DIS
LIN {X -91.3988,Y 108.5744,Z 186,A 130.8576,B 2.821,C 0.0605,E1 2.7221,E2 322.9476} C_DIS
LIN {X -87.8671,Y 111.4519,Z 186,A 128.94,B 2.821,C 0.0577,E1 2.7263,E2 324.8737} C_DIS
LIN {X -84.3232,Y 114.157,Z 186,A 127.0749,B 2.821,C 0.0551,E1 2.7305,E2 326.7456} C_DIS
LIN {X -80.5145,Y 116.8742,Z 186,A 125.1714,B 2.8212,C 0.0523,E1 2.7349,E2 328.6497} C_DIS
LIN {X -77.0678,Y 119.1752,Z 186,A 123.4706,B 2.8212,C 0.05,E1 2.7389,E2 330.3527} C_DIS
LIN {X -73.1683,Y 121.6084,Z 186,A 121.4314,B 2.8212,C 0.0483,E1 2.7438,E2 332.4137} C_DIS
LIN {X -69.7117,Y 123.6221,Z 186,A 119.8723,B 2.8212,C 0.046,E1 2.7476,E2 333.9647} C_DIS
LIN {X -65.671,Y 125.8132,Z 186,A 118.0502,B 2.8213,C 0.0436,E1 2.752,E2 335.7813} C_DIS
LIN {X -60.8471,Y 128.2158,Z 186,A 115.8864,B 2.8213,C 0.0411,E1 2.7575,E2 337.9422} C_DIS
LIN {X -57.6952,Y 129.6645,Z 186,A 114.4514,B 2.8213,C 0.0398,E1 2.7611,E2 339.3806} C_DIS
LIN {X -54.4376,Y 131.0654,Z 186,A 112.9655,B 2.8213,C 0.0386,E1 2.765,E2 340.8723} C_DIS
LIN {X -50.534,Y 132.6217,Z 186,A 110.7124,B 2.8213,C 0.04,E1 2.771,E2 343.1936} C_DIS
LIN {X -46.1763,Y 134.1991,Z 186,A 109.3515,B 2.8214,C 0.0358,E1 2.7744,E2 344.4901} C_DIS
LIN {X -42.3212,Y 135.4664,Z 186,A 107.7191,B 2.8214,C 0.0346,E1 2.7788,E2 346.1209} C_DIS
LIN {X -39.2309,Y 136.3927,Z 186,A 106.0798,B 2.8214,C 0.0355,E1 2.7833,E2 347.8012} C_DIS
LIN {X -35.9504,Y 137.2937,Z 186,A 105.025,B 2.8214,C 0.033,E1 2.786,E2 348.8157} C_DIS
LIN {X -32.8892,Y 138.0581,Z 186,A 103.7288,B 2.8214,C 0.0324,E1 2.7896,E2 350.1139} C_DIS
LIN {X -29.0062,Y 138.9272,Z 186,A 101.9692,B 2.8214,C 0.0325,E1 2.7944,E2 351.8918} C_DIS
LIN {X -22.4508,Y 140.1361,Z 186,A 99.197,B 2.8214,C 0.0321,E1 2.8021,E2 354.6727} C_DIS
LIN {X -17.7543,Y 140.808,Z 186,A 97.3492,B 2.8214,C 0.0312,E1 2.8072,E2 356.5111} C_DIS
LIN {X -13.6721,Y 141.2612,Z 186,A 95.7577,B 2.8214,C 0.0305,E1 2.8116,E2 358.0935} C_DIS
LIN {X -9.4176,Y 141.6102,Z 186,A 93.8888,B 2.8214,C 0.0313,E1 2.8168,E2 359.9797} C_DIS
LIN {X -5.7559,Y 141.8048,Z 186,A 92.5355,B 2.8214,C 0.0305,E1 2.8206,E2 361.3165} C_DIS
LIN {X -1.6738,Y 141.9132,Z 186,A 90.7945,B 2.8214,C 0.0313,E1 2.8255,E2 363.0683} C_DIS
LIN {X 2.4263,Y 141.9007,Z 186,A 89.2797,B 2.8214,C 0.0306,E1 2.8297,E2 364.5649} C_DIS
LIN {X 6.5276,Y 141.7724,Z 186,A 87.5147,B 2.8214,C 0.0317,E1 2.8346,E2 366.3429} C_DIS
LIN {X 10.8556,Y 141.5065,Z 186,A 85.7767,B 2.8214,C 0.0322,E1 2.8395,E2 368.0786} C_DIS
LIN {X 15.2688,Y 141.0975,Z 186,A 84.1201,B 2.8214,C 0.0322,E1 2.844,E2 369.718} C_DIS
LIN {X 18.5703,Y 140.7011,Z 186,A 82.835,B 2.8214,C 0.0324,E1 2.8476,E2 370.9955} C_DIS
LIN {X 22.1433,Y 140.1838,Z 186,A 81.3215,B 2.8214,C 0.0336,E1 2.8518,E2 372.5156} C_DIS
LIN {X 25.5099,Y 139.6106,Z 186,A 79.9391,B 2.8214,C 0.0344,E1 2.8556,E2 373.898} C_DIS
LIN {X 28.9059,Y 138.9476,Z 186,A 78.635,B 2.8214,C 0.0348,E1 2.8591,E2 375.1901} C_DIS
LIN {X 32.1115,Y 138.2415,Z 186,A 77.2412,B 2.8214,C 0.0362,E1 2.863,E2 376.5921} C_DIS
LIN {X 37.1079,Y 136.985,Z 186,A 75.3149,B 2.8214,C 0.0369,E1 2.8681,E2 378.4987} C_DIS
LIN {X 42.9878,Y 135.254,Z 186,A 72.3267,B 2.8214,C 0.0429,E1 2.8763,E2 381.5504} C_DIS
LIN {X 47.3929,Y 133.7762,Z 186,A 71.0035,B 2.8214,C 0.0408,E1 2.8796,E2 382.8044} C_DIS
LIN {X 50.4593,Y 132.6497,Z 186,A 69.6836,B 2.8214,C 0.0423,E1 2.8831,E2 384.1242} C_DIS
LIN {X 53.3607,Y 131.5077,Z 186,A 68.4567,B 2.8214,C 0.0435,E1 2.8862,E2 385.3467} C_DIS
LIN {X 56.6427,Y 130.1278,Z 186,A 67.0433,B 2.8213,C 0.0451,E1 2.8899,E2 386.7569} C_DIS
LIN {X 59.9006,Y 128.6607,Z 186,A 65.6217,B 2.8213,C 0.0468,E1 2.8935,E2 388.1758} C_DIS
LIN {X 63.2961,Y 127.0254,Z 186,A 64.1284,B 2.8213,C 0.0486,E1 2.8972,E2 389.6654} C_DIS
LIN {X 67.3073,Y 124.9474,Z 186,A 62.2827,B 2.8212,C 0.0514,E1 2.9018,E2 391.5138} C_DIS
LIN {X 71.2428,Y 122.746,Z 186,A 60.508,B 2.8212,C 0.0537,E1 2.9061,E2 393.2825} C_DIS
LIN {X 75.0929,Y 120.4291,Z 186,A 58.7836,B 2.8211,C 0.0558,E1 2.9102,E2 394.9956} C_DIS
LIN {X 78.5856,Y 118.1798,Z 186,A 57.1598,B 2.8211,C 0.0581,E1 2.9139,E2 396.6126} C_DIS
LIN {X 81.993,Y 115.8416,Z 186,A 55.4831,B 2.821,C 0.061,E1 2.9178,E2 398.2904} C_DIS
LIN {X 85.7775,Y 113.0683,Z 186,A 53.6595,B 2.821,C 0.0638,E1 2.9219,E2 400.1051} C_DIS
LIN {X 89.395,Y 110.2305,Z 186,A 51.9477,B 2.8209,C 0.066,E1 2.9256,E2 401.7987} C_DIS
LIN {X 92.3627,Y 107.7559,Z 186,A 50.3347,B 2.8208,C 0.0694,E1 2.929,E2 403.4185} C_DIS
LIN {X 95.7378,Y 104.769,Z 186,A 48.4937,B 2.8207,C 0.0732,E1 2.9328,E2 405.2624} C_DIS
LIN {X 99.5349,Y 101.1679,Z 186,A 46.5846,B 2.8207,C 0.0757,E1 2.9366,E2 407.1459} C_DIS
LIN {X 102.526,Y 98.1352,Z 186,A 44.8921,B 2.8205,C 0.079,E1 2.9399,E2 408.8352} C_DIS
LIN {X 105.6533,Y 94.7602,Z 186,A 43.1199,B 2.8205,C 0.0823,E1 2.9432,E2 410.5969} C_DIS
LIN {X 108.5359,Y 91.4447,Z 186,A 41.4361,B 2.8203,C 0.0854,E1 2.9463,E2 412.2696} C_DIS
LIN {X 111.2745,Y 88.092,Z 186,A 39.6692,B 2.8203,C 0.0895,E1 2.9494,E2 414.0393} C_DIS
LIN {X 114.0535,Y 84.4632,Z 186,A 37.9469,B 2.8201,C 0.0926,E1 2.9523,E2 415.7463} C_DIS
LIN {X 116.7223,Y 80.7351,Z 186,A 36.1694,B 2.82,C 0.0963,E1 2.9551,E2 417.5149} C_DIS
LIN {X 119.1656,Y 77.0825,Z 186,A 34.4859,B 2.8199,C 0.0997,E1 2.9577,E2 419.1872} C_DIS
LIN {X 121.4777,Y 73.3844,Z 186,A 32.8085,B 2.8197,C 0.1032,E1 2.9601,E2 420.8544} C_DIS
LIN {X 123.6961,Y 69.5799,Z 186,A 31.0866,B 2.8197,C 0.1071,E1 2.9625,E2 422.5697} C_DIS
LIN {X 125.8129,Y 65.6716,Z 186,A 29.4515,B 2.8195,C 0.1101,E1 2.9646,E2 424.1848} C_DIS
LIN {X 127.3924,Y 62.5521,Z 186,A 28.0928,B 2.8194,C 0.1132,E1 2.9663,E2 425.5372} C_DIS
LIN {X 128.9842,Y 59.2009,Z 186,A 26.6507,B 2.8192,C 0.1166,E1 2.968,E2 426.9726} C_DIS
LIN {X 130.4678,Y 55.8564,Z 186,A 25.2566,B 2.8192,C 0.1196,E1 2.9695,E2 428.3566} C_DIS
LIN {X 131.9236,Y 52.3291,Z 186,A 23.7887,B 2.819,C 0.123,E1 2.9711,E2 429.8157} C_DIS
LIN {X 132.9811,Y 49.5745,Z 186,A 22.644,B 2.8188,C 0.1257,E1 2.9722,E2 430.9548} C_DIS
LIN {X 134.1918,Y 46.1975,Z 186,A 21.2419,B 2.8187,C 0.1292,E1 2.9735,E2 432.3516} C_DIS
LIN {X 135.1856,Y 43.2019,Z 186,A 20.0134,B 2.8185,C 0.1322,E1 2.9746,E2 433.5747} C_DIS
LIN {X 136.5212,Y 38.7798,Z 186,A 18.3702,B 2.8185,C 0.1351,E1 2.9758,E2 435.1898} C_DIS
LIN {X 137.1667,Y 36.4266,Z 186,A 17.3122,B 2.8182,C 0.1385,E1 2.9766,E2 436.2578} C_DIS
LIN {X 138.1006,Y 32.7129,Z 186,A 15.834,B 2.8181,C 0.1421,E1 2.9776,E2 437.728} C_DIS
LIN {X 138.9351,Y 28.9671,Z 186,A 14.1603,B 2.8178,C 0.1475,E1 2.9786,E2 439.4188} C_DIS
Enddeposition()
END
